		(*####################  DEBUG-MESSAGE  ###################################*)
		(*IF _debug_enable THEN
			LOG_CL.NEW_MSG := 'Repeat request after waittime / Part ~2 / Count ~3';
			LOG_CL.PRINTF[2] := INT_TO_STRING(cycle);
			LOG_CL.PRINTF[3] := USINT_TO_STRING(repeat_count);
			LOG_MSG();
		END_IF;*)
		(*########################################################################*)

		repeat_request := FALSE;
		state := 50;

	END_IF;

END_CASE;

(* ---------------- DNS --------------- *)
DNS_CLIENT(	IP_C:=IP_C,
			S_BUF:=S_BUF,
			R_BUF:=R_BUF,
			DOMAIN:=URL_DATA.DOMAIN,
			IP4_DNS:=DWORD#00,
			ACTIVATE:=state=40 (* DNS Start *)
			);
(* nicht oder nicht direkt verwendete Parameter *)
(*	DWORD :=DNS_CLIENT.IP4;
	BOOL  :=DNS_CLIENT.DONE;
	BYTE  :=DNS_CLIENT.ERROR; *)
(* -------------------------------------*)

(* ------------- HTTP_GET --------------- *)
HTTP_GET(	IP_C:=IP_C,
			S_BUF:=S_BUF,
			R_BUF:=R_BUF,
			IP4:=DNS_CLIENT.IP4,
			GET:=state=60,
			MODE:=BYTE#2, (* HTTP 1.1 mit persistenter Verbindung *)
			UNLOCK_BUF:=state=100,
			URL_DATA:=URL_DATA
			);

(* nicht oder nicht direkt verwendete Parameter *)
(*	STRING := HTTP_GET.HTTP_STATUS;
	UINT :=HTTP_GET.HEADER_START;
	UINT :=HTTP_GET.HEADER_STOP;
	UINT :=HTTP_GET.BODY_START;
	UINT :=HTTP_GET.BODY_STOP;
	BOOL :=HTTP_GET.DONE;
	BYTE :=HTTP_GET.ERROR;
*)
(* -------------------------------------*)

activate_last := ACTIVATE;

(*####################  DEBUG-MESSAGE  ###################################*)
(*IF _debug_enable THEN
	IF state <> _debug_state_last THEN
		LOG_CL.NEW_MSG := 'yw-step: /last ~1 /New ~2';
		LOG_CL.PRINTF[1] := INT_TO_STRING(_debug_state_last);
		LOG_CL.PRINTF[2] := INT_TO_STRING(state);
		LOG_MSG();
		_debug_state_last := state;
	END_IF;
END_IF;*)
(*########################################################################*)

(* revision history
ks	18. dez. 2008	rev 1.0
	original version

ks	01. oct. 2009	rev 1.1
	YAHOO_WEATHER_DATA

ks	24. sep. 2010	rev 1.2
	new URL-Location-parameter and REAL_CHECK (TwinCat BUG) 

ks	04. may. 2011	rev 1.3
	neue elemente:  CUR_CONDITIONS_ICON, FORCAST_TODAY_ICON, FORCAST_TOMORROW_ICON

ks	30. mar. 2016	rev 1.4
	änderung der api schnittstelle (URL) von yahoo

ks	01. jun. 2016	rev 1.5
	komplette überarbeitung auf neue yahoo-api

ks	22. may. 2017	rev 1.6
	automatische wiederholung der Abfrage wenn keine Daten vorhanden sind
*)

END_FUNCTION_BLOCK

// POUs/OTHER/XML_READER
FUNCTION_BLOCK XML_READER
VAR_IN_OUT
	CTRL : XML_CONTROL;
	BUF : NW_BUF_LONG;
END_VAR
VAR
	index :	INT;
	index2 : INT;
	stop : INT;
	mode : INT;
	command : WORD;
	c :	BYTE;
	s1 : INT;
	e1 : INT;
	path_overflow : BOOL;
	empty_tag : BOOL;
	s_code : STRING(10);
	e_code : STRING(10);
	watchdog : TON;

	(*LOG_MSG : LOG_MSG;
	_debug_enable : BOOL := TRUE;*)

END_VAR

(*

version 1.2		10. mai 2010
programmer 	ks
tested by		ks

XML_READER ermöglicht das serielle Parsen und die Auswertung von XML_Elementen in einem Buffer
*)

(*

TYP
00 = UNBEKANNT
01 = ELEMENT (STANDARD)
02 = CLOSE ELEMENT 
03 = TEXT
04 = ATTRIBUTE
05 = ELEMENT (PROCESSING INSTRUCTION) 

12 = !CDATA
13 = !COMMENT
14 = !DTD ELEMENT (Document Type Declarations )

98 = WATCHDOG
99 = ENDE

Bei Typ 02 werden keine Blockdaten ausgegeben !

*)

(* ---------- Init -------------- *)
IF OSCAT_BASIC.BIT_OF_DWORD(WORD_TO_DWORD(CTRL.COMMAND),15) THEN
	COMMAND := CTRL.COMMAND;
	CTRL.COMMAND := WORD#0;

	index := UINT_TO_INT(CTRL.START_POS);
	stop := UINT_TO_INT(CTRL.STOP_POS);
	mode := 100;
	path_overflow := FALSE;

	CTRL.TYP := 0;
	CTRL.COUNT := UINT#00;
	CTRL.LEVEL := UINT#00;
	CTRL.ATTRIBUTE := '';
	CTRL.ELEMENT := '';
	CTRL.PATH := '';
	CTRL.VALUE := '';

	WATCHDOG.PT := CTRL.WATCHDOG;
END_IF;

(*----------------------------------------------- *)

IF index < 0 THEN RETURN;END_IF;

CTRL.BLOCK1_START := UINT#0;
CTRL.BLOCK1_STOP := UINT#0;
CTRL.BLOCK2_START := UINT#0;
CTRL.BLOCK2_STOP := UINT#0;

WATCHDOG(IN:=FALSE); (* Timer stoppen *)

WHILE (TRUE) DO

	(* -------------- WATCHDOG ------------------ *)
	WATCHDOG(IN:=CTRL.WATCHDOG > T#0s);
	IF WATCHDOG.Q THEN
		CTRL.TYP := 98;
    		(*####################  DEBUG-MESSAGE  ###################################*)
    		(*IF _debug_enable THEN
      			LOG_CL.NEW_MSG := 'WATCHDOG:';
      			LOG_MSG();
    		END_IF;*)
    		(*########################################################################*)
		RETURN;
	END_IF;

	(* -------------- PARSING END ------------------ *)
	IF index > stop THEN
		CTRL.COUNT := CTRL.COUNT + UINT#1;
		CTRL.TYP := 99;
    		(*####################  DEBUG-MESSAGE  ###################################*)
    		(*IF _debug_enable THEN
      			LOG_CL.NEW_MSG := 'EX: #T:~1 #C:~2 #P:~6 #L:~7';
      			LOG_CL.PRINTF[1] := INT_TO_STRING(CTRL.TYP);
      			LOG_CL.PRINTF[2] := UINT_TO_STRING(CTRL.COUNT);
      			LOG_CL.PRINTF[6] := CTRL.PATH;
      			LOG_CL.PRINTF[7] := UINT_TO_STRING(CTRL.LEVEL);
      			LOG_MSG();
    		END_IF;*)
    		(*########################################################################*)
		mode  := 0; (* Schritt ruecksetzen *)
		index := 0; (* Abarbeitung stoppen *)
		RETURN;
	END_IF;

	CASE mode OF

	100: (* ---------- ELEMENT SECTION ------------------ *)
		(* search begin of element *)
		s1 := 0;
		e1 := 0;
		WHILE (index <= stop) DO
			IF BUF[INDEX]=BYTE#60 THEN (* '<' TagBegin *)
				index := index + 1;
				C := BUF[index];
				IF C = BYTE#47 THEN (* '/' TagTerm *)
					mode := 300; (* End Element Section *)
				ELSIF C = BYTE#33 THEN (* '!' for Special Section *)
					index := index + 1;
					mode := 500;
				ELSE
					s1 := index;
				END_IF;
				EXIT;
			END_IF;
			index := index + 1;
		END_WHILE;

		(* analyse element *)
		CTRL.TYP := 0; (* TYP löschen *)
		IF s1 > 0 THEN
			WHILE (index <= stop AND e1 = 0) DO
				c := BUF[index];
				(* whitespace zeichen = Element with Attributes *)
				IF c <= BYTE#32 THEN
					(* suche nächstes druckbares zeichen *)
					index2 := index;
					WHILE (index2 <= stop) AND (BUF[index2] <= BYTE#32) DO
						index2 := index2 + 1;
					END_WHILE;
					IF BUF[index2] = BYTE#47 THEN (* pruefe auf leeres Element '/' *)
						index := index2;
						e1 := index - 2;
						CTRL.TYP := 1; (* struktur-element *)
						mode := 300;   (* Close Element *)
						EXIT;
					END_IF;

					e1 := index - 1;
					CTRL.TYP := 1; (* Element mit Attribute *)
					mode := 400;

				ELSIF c = BYTE#62 THEN (* '>' TagEnd *)

					(* pruefe auf leeres Element <xx/> *)
					index2 := index - 1;
					IF BUF[index2] = BYTE#47 THEN (* TagTerm '/' *)
						e1 := index2 - 1;
						CTRL.TYP := 1;
						EMPTY_TAG := TRUE; (* EMPTY TAG Mode *)
						mode := 200; (* TEXT Element *)
						EXIT;
					END_IF;

					e1 := index - 1;
					index2 := index + 1;

					(* untersuche nachfolgendes Element *)
					WHILE (index2 <= stop) DO
						c := BUF[index2];
						IF c = BYTE#60 THEN (* '<' TagBegin *)

							index2 := index2 + 1; (* geht bei PCWORX leider nicht anders !*)
							c := BUF[index2];
							index2 := index2 - 1;
							IF c = BYTE#47 THEN (* TagTerm '/' *)
								empty_tag := TRUE;
								mode := 200; (* TEXT Element *)
							ELSE
								mode := 100; (* Element *)
							END_IF;
							CTRL.TYP := 1; (* struktur-element *)
							EXIT;
						ELSIF c > BYTE#32  THEN (* Printable-Character *)
							CTRL.TYP := 1; (* element with text *)
							mode := 200;
							EXIT;
						END_IF;
						index2 := index2 + 1;
					END_WHILE;
				END_IF;
				index := index + 1;
			END_WHILE;
		END_IF;

		(* Neues Element gefunden*)
		IF CTRL.TYP > 0 THEN

			(* Sonderprüfung auf Processing Instruction (PI) *)
			IF BUF[s1] = BYTE#63 THEN (* '?' for Processing Instruction *)
				s1 := s1 + 1; (* führendes '?' auslassen *)
				CTRL.TYP := 5;
			END_IF;
			CTRL.BLOCK1_START := INT_TO_UINT(s1);
			CTRL.BLOCK1_STOP  := INT_TO_UINT(e1);
			CTRL.ELEMENT := OSCAT_BASIC.BUFFER_TO_STRING(PT:=ADR(BUF),SIZE:=INT_TO_UINT(stop + 1),START:=CTRL.BLOCK1_START,STOP:=CTRL.BLOCK1_STOP);
			CTRL.COUNT := CTRL.COUNT + UINT#1;
			CTRL.LEVEL := CTRL.LEVEL + UINT#1;

			IF path_overflow = FALSE THEN
				(* Stringlänge überwachen *)
				IF LEN(CTRL.PATH) + LEN(CTRL.ELEMENT) + 1 > 250 THEN
					path_overflow := TRUE;
					CTRL.PATH := 'OVERFLOW';
				ELSE
					CTRL.PATH := CONCAT(CTRL.PATH,'/');
					CTRL.PATH  := CONCAT(CTRL.PATH,CTRL.ELEMENT);
				END_IF;
			END_IF;

			IF OSCAT_BASIC.BIT_OF_DWORD(WORD_TO_DWORD(COMMAND),CTRL.TYP) THEN
        				(*####################  DEBUG-MESSAGE  ###################################*)
        				(*IF _debug_enable THEN
          				LOG_CL.NEW_MSG := 'EL: #T:~1 #C:~2 #E:~3 #P:~6 #L:~7';
          				LOG_CL.PRINTF[1] := INT_TO_STRING(CTRL.TYP);
          				LOG_CL.PRINTF[2] := UINT_TO_STRING(CTRL.COUNT);
          				LOG_CL.PRINTF[3] := CTRL.ELEMENT;
          				LOG_CL.PRINTF[6] := CTRL.PATH;
          				LOG_CL.PRINTF[7] := UINT_TO_STRING(CTRL.LEVEL);
          				LOG_MSG();
        				END_IF;*)
        				(*########################################################################*)
				RETURN;
			END_IF;
		END_IF;

	200: (* ---------- TEXT SECTION ------------------ *)
		CTRL.VALUE := '';
		IF empty_tag = FALSE THEN
			s1 := index;
			(* suche '<' EndTag*)
			WHILE (index <= stop) AND (BUF[index] <> BYTE#60) DO
				index := index + 1;
			END_WHILE;

			E1 := index - 1;
			CTRL.BLOCK1_START := INT_TO_UINT(s1);
			CTRL.BLOCK1_STOP  := INT_TO_UINT(e1);
			CTRL.VALUE := OSCAT_BASIC.BUFFER_TO_STRING(PT:=ADR(BUF),SIZE:=INT_TO_UINT(stop + 1),START:=CTRL.BLOCK1_START,STOP:=CTRL.BLOCK1_STOP);
		END_IF;

		empty_tag := FALSE;
		mode := 300; (* -> NEXT-JOB: END ELEMENT *)
		CTRL.COUNT := CTRL.COUNT + UINT#1;
		CTRL.TYP := 3;

		IF OSCAT_BASIC.BIT_OF_DWORD(WORD_TO_DWORD(command),CTRL.TYP) THEN
      			(*####################  DEBUG-MESSAGE  ###################################*)
      			(*IF _debug_enable THEN
        				LOG_CL.NEW_MSG := 'TE: #T:~1 #C:~2 #E:~3 #V:~4 #P:~6 #L:~7';
        				LOG_CL.PRINTF[1] := INT_TO_STRING(CTRL.TYP);
        				LOG_CL.PRINTF[2] := UINT_TO_STRING(CTRL.COUNT);
        				LOG_CL.PRINTF[3] := CTRL.ELEMENT;
        				LOG_CL.PRINTF[4] := CTRL.VALUE;
        				LOG_CL.PRINTF[6] := CTRL.PATH;
        				LOG_CL.PRINTF[7] := UINT_TO_STRING(CTRL.LEVEL);
        				LOG_MSG();
      			END_IF;*)
      			(*########################################################################*)
			RETURN;
		END_IF;

	300: (* ---------- END ELEMENT SECTION ------------------ *)
		WHILE (index <= stop) DO
			c := BUF[index];
			IF c = BYTE#62 THEN (* '>' TagEnd *)
				index := index + 1;
				s1 := OSCAT_BASIC.FINDB(str1:=CTRL.PATH,str2:='/');
				IF path_overflow = FALSE THEN
					IF s1 > 1 THEN
						CTRL.ELEMENT := RIGHT(CTRL.PATH,LEN(CTRL.PATH) - s1);
						CTRL.PATH := LEFT(CTRL.PATH,s1 - 1);
					ELSE
						CTRL.ELEMENT := RIGHT(CTRL.PATH,LEN(CTRL.PATH) - 1);
						CTRL.PATH :='';
					END_IF;
				END_IF;

				CTRL.LEVEL := CTRL.LEVEL - UINT#1;
				CTRL.COUNT := CTRL.COUNT + UINT#1;
				CTRL.TYP := 2;
				mode := 100;

				IF OSCAT_BASIC.BIT_OF_DWORD(WORD_TO_DWORD(COMMAND),CTRL.TYP) THEN
         	 				(*####################  DEBUG-MESSAGE  ###################################*)
          				(*IF _debug_enable THEN
            					LOG_CL.NEW_MSG := 'CE: #T:~1 #C:~2 #E:~3 #P:~6 #L:~7';
            					LOG_CL.PRINTF[1] := INT_TO_STRING(CTRL.TYP);
            					LOG_CL.PRINTF[2] := UINT_TO_STRING(CTRL.COUNT);
            					LOG_CL.PRINTF[3] := CTRL.ELEMENT;
            					LOG_CL.PRINTF[6] := CTRL.PATH;
            					LOG_CL.PRINTF[7] := UINT_TO_STRING(CTRL.LEVEL);
            					LOG_MSG();
          				END_IF;*)
          				(*########################################################################*)
					RETURN;
				ELSE
					EXIT;
				END_IF;
			END_IF;
			index := index + 1;
		END_WHILE;

	400: (* ---------- ATTRIBUTE SECTION ------------------ *)
		(* search first normal charakter *)
		WHILE (index <= stop AND BUF[index] <= BYTE#32) DO
			index := index + 1;
		END_WHILE;

		(* begin Attribe name *)
		e1 := 0;
		s1 := index;
		(* search end of Attrib Name '=' *)
		WHILE (index <= stop) DO
			IF BUF[index] = BYTE#61 THEN (* '=' Equals *)
				e1 := index - 1;
				EXIT;
			END_IF;
			index := index + 1;
		END_WHILE;

		IF e1 > 0 THEN
			(* Attribute Name *)
			CTRL.BLOCK1_START := INT_TO_UINT(s1);
			CTRL.BLOCK1_STOP  := INT_TO_UINT(e1);
			CTRL.ATTRIBUTE := OSCAT_BASIC.BUFFER_TO_STRING(PT:=ADR(BUF),SIZE:=INT_TO_UINT(STOP + 1),START:=CTRL.BLOCK1_START,STOP:=CTRL.BLOCK1_STOP);
			(* search end of Attrib Value '=' *)
			index := index + 2;
			e1 := 0;
			s1 := INDEX;
			WHILE (index <= stop AND e1 = 0) DO
				c := BUF[index];
				IF c = BYTE#34 OR c = BYTE#39 THEN (* " OR ' Equals *)
					e1 := index - 1;
				END_IF;
				index := index + 1;
			END_WHILE;

			IF e1 > 0 THEN
				(* Value *)
				CTRL.BLOCK2_START := INT_TO_UINT(s1);
				CTRL.BLOCK2_STOP  := INT_TO_UINT(e1);

				(* bei leeren "" ist start groesser als stop und wird somit zum leerstring *)
				CTRL.VALUE := OSCAT_BASIC.BUFFER_TO_STRING(PT:=ADR(BUF),SIZE:=INT_TO_UINT(stop + 1),START:=CTRL.BLOCK2_START,STOP:=CTRL.BLOCK2_STOP);
				(* search next non white space charakter *)
				WHILE (index <= stop AND BUF[index] <= BYTE#32) DO
					index := index + 1;
				END_WHILE;

					c := BUF[index];
					(* TagEnd '>' *)
					IF c = BYTE#62 THEN
						index := index + 1;
						index2 := index;

					(* search next non white space charakter *)
					WHILE (index <= stop AND BUF[index] <= BYTE#32) DO
						index := index + 1;
					END_WHILE;

					IF BUF[index] = BYTE#60 THEN (* TagBegin '<' *)
						mode := 100; (* -> NEXT-JOB: ELEMENT-SECTION *)
					ELSE
						index := index2;
						mode := 200; (* -> NEXT-JOB: TEXT-SECTION *)
					END_IF;

				ELSIF c = BYTE#47 OR c = BYTE#63 THEN (* TagTerm '/' OR '?' end Processing Instruction *)
					mode := 300; (* -> NEXT-JOB: END ELEMENT *)
				ELSE
					mode := 400; (* -> NEXT-JOB: ATTRIBUTE-SECTION *)
				END_IF;

				CTRL.COUNT := CTRL.COUNT + UINT#1;
				CTRL.TYP := 4;
				IF OSCAT_BASIC.BIT_OF_DWORD(WORD_TO_DWORD(command),CTRL.TYP) THEN
          				(*####################  DEBUG-MESSAGE  ###################################*)
          				(*IF _debug_enable THEN
            					LOG_CL.NEW_MSG := 'AT: #T:~1 #C:~2 #E:~3 #A:~4 #V:~5 #P:~6 #L:~7';
            					LOG_CL.PRINTF[1] := INT_TO_STRING(CTRL.TYP);
            					LOG_CL.PRINTF[2] := UINT_TO_STRING(CTRL.COUNT);
            					LOG_CL.PRINTF[3] := CTRL.ELEMENT;
            					LOG_CL.PRINTF[4] := CTRL.ATTRIBUTE;
            					LOG_CL.PRINTF[5] := CTRL.VALUE;
            					LOG_CL.PRINTF[6] := CTRL.PATH;
            					LOG_CL.PRINTF[7] := UINT_TO_STRING(CTRL.LEVEL);
            					LOG_MSG();
          				END_IF;*)
          				(*########################################################################*)
					RETURN;
				END_IF;
			END_IF;
		END_IF;

	500: (* ---------- SPECIAL DATA SECTION (Document Type Declarations) ---------- *)

		CTRL.TYP := 0;
		s1 := 0;
		index2 := 11;

		WHILE (s1 = 0) DO
			index2 := index2 + 1;
			CTRL.TYP := index2;

			CASE index2 OF
			12: (* CDATA *)
				s_code := '[CDATA[';
				e_code := ']]>';
			13: (* COMMENT *)
				s_code := '--';
				e_code := '-->';
			14: (* ANY DTD *)
				e_code := '';
				s1 := index;
				EXIT;
			END_CASE;

			e1 := LEN(s_code);
			IF OSCAT_BASIC.BUFFER_SEARCH(PT:=ADR(BUF),SIZE:=INT_TO_UINT(index + e1),STR:=S_CODE,POS:=index,IGN:=FALSE) = INDEX THEN
				s1 := index + e1;
			END_IF;
		END_WHILE;

		CTRL.BLOCK1_START := INT_TO_UINT(s1);
		IF LEN(e_code) > 0 THEN
			(* Ende Kennung suchen *)
			e1 := OSCAT_BASIC.BUFFER_SEARCH(PT:=ADR(BUF),SIZE:=INT_TO_UINT(stop + 1),STR:=e_code,POS:=index,IGN:=FALSE);
			CTRL.BLOCK1_STOP := INT_TO_UINT(e1 - 1);
			index := e1 + LEN(e_code); (* naechstes element *)
		ELSE
			(* suche '>' EndTag*)
			index2 := 1; (* <> Paar zähler *)
			WHILE (index <= stop AND index2 > 0) DO
				c := BUF[index];
				IF c = BYTE#60 THEN (* '<' TagBegin *)
					index2 := index2 + 1;
				ELSIF c = BYTE#62 THEN (* '>' TagEnd   *)
					index2 := index2 - 1;
				ELSIF c = BYTE#34 OR c = BYTE#39 THEN (* " Double Quote OR ' Single Quote *)
					index := index + 1;
					WHILE (index <= stop) DO
						c := BUF[index];
						IF c = BYTE#34 OR c = BYTE#39 THEN (* " Double Quote OR ' Single Quote *)
							EXIT;
						END_IF;
						index := index + 1;
					END_WHILE;
				END_IF;
				index := index + 1;
			END_WHILE;
			CTRL.BLOCK1_STOP := INT_TO_UINT(index - 2);
		END_IF;

		CTRL.VALUE := OSCAT_BASIC.BUFFER_TO_STRING(PT:=ADR(BUF),SIZE:=INT_TO_UINT(stop + 1),START:=CTRL.BLOCK1_START,STOP:=CTRL.BLOCK1_STOP);
		CTRL.COUNT := CTRL.COUNT + UINT#1;
		mode := 100; (* -> NEXT-JOB: ELEMENT *)

		IF OSCAT_BASIC.BIT_OF_DWORD(WORD_TO_DWORD(command),CTRL.TYP) THEN
      			(*####################  DEBUG-MESSAGE  ###################################*)
      			(*IF _debug_enable THEN
        				LOG_CL.NEW_MSG := 'DTD: #T:~1 #C:~2 #S:~3 #E:~4 #V:~5 #P:~6 #L:~7';
        				LOG_CL.PRINTF[1] := INT_TO_STRING(CTRL.TYP);
        				LOG_CL.PRINTF[2] := UINT_TO_STRING(CTRL.COUNT);
        				LOG_CL.PRINTF[3] := UINT_TO_STRING(CTRL.BLOCK1_START);
        				LOG_CL.PRINTF[4] := UINT_TO_STRING(CTRL.BLOCK1_STOP);
        				LOG_CL.PRINTF[5] := CTRL.VALUE;
        				LOG_CL.PRINTF[6] := CTRL.PATH;
        				LOG_CL.PRINTF[7] := UINT_TO_STRING(CTRL.LEVEL);
        				LOG_MSG();
      			END_IF;*)
      			(*########################################################################*)
			RETURN;
		END_IF;

	END_CASE;
END_WHILE;


(* revision history
ks	18. oct. 2008	rev 1.0
	original version

ks	20. oct. 2009	rev 1.1
	Networkbuffer und Buffer-funktionen auf Basis 0

ks	10. mai. 2010	rev 1.2
	stringlänge maximal 250 zeichen

*)

END_FUNCTION_BLOCK

// POUs/DEMO/DNS_DYN_DEMO
PROGRAM DNS_DYN_DEMO
VAR
	DNS_DYN : DNS_DYN;
	IP_C : IP_C;
	S_BUF : NETWORK_BUFFER;
	R_BUF : NETWORK_BUFFER;
	IP_CONTROL : IP_CONTROL;
	enable: BOOL;
	done : BOOL;
	error_c : DWORD;
	error_t : BYTE;
	busy : BOOL;
	COUNT_DR: oscat_basic.COUNT_DR;
	z: DWORD;

	GET_WAN_IP : GET_WAN_IP;
	t1: TON;
	done2 : BOOL;
	error_c2 : DWORD;
	error_t2 : BYTE;
	update : BOOL;
	new_ip: BOOL;
	wan_ip4: DWORD;
END_VAR
VAR // added by the converter: edge detectors and wires of the graphical bodies
    _w1 : ANY;
END_VAR

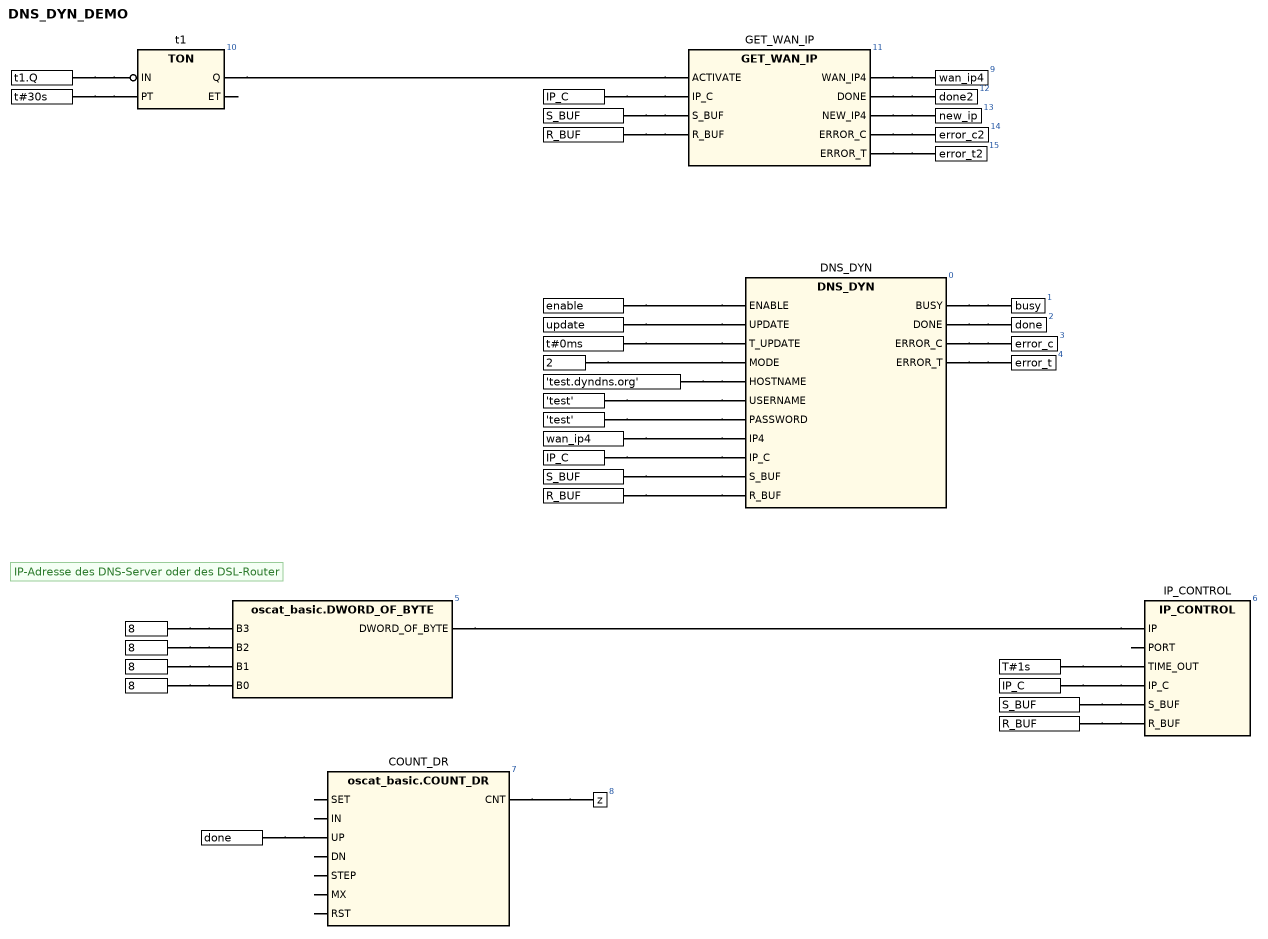
DNS_DYN(
    ENABLE := enable,
    UPDATE := update,
    T_UPDATE := t#0ms,
    MODE := 2,
    HOSTNAME := 'test.dyndns.org',
    USERNAME := 'test',
    PASSWORD := 'test',
    IP4 := wan_ip4,
    IP_C := IP_C,
    S_BUF := S_BUF,
    R_BUF := R_BUF);
busy := DNS_DYN.BUSY;
done := DNS_DYN.DONE;
error_c := DNS_DYN.ERROR_C;
error_t := DNS_DYN.ERROR_T;
// IP-Adresse des DNS-Server oder des DSL-Router
_w1 := oscat_basic.DWORD_OF_BYTE(B3 := 8, B2 := 8, B1 := 8, B0 := 8);
IP_CONTROL(IP := _w1, TIME_OUT := T#1s, IP_C := IP_C, S_BUF := S_BUF, R_BUF := R_BUF);
COUNT_DR(UP := done); // oscat_basic.COUNT_DR
z := COUNT_DR.CNT;
wan_ip4 := GET_WAN_IP.WAN_IP4;
t1(IN := NOT t1.Q, PT := t#30s); // TON
GET_WAN_IP(ACTIVATE := t1.Q, IP_C := IP_C, S_BUF := S_BUF, R_BUF := R_BUF);
done2 := GET_WAN_IP.DONE;
new_ip := GET_WAN_IP.NEW_IP4;
error_c2 := GET_WAN_IP.ERROR_C;
error_t2 := GET_WAN_IP.ERROR_T;

END_PROGRAM

// POUs/NETWORK/GET_WAN_IP
FUNCTION_BLOCK GET_WAN_IP
VAR_IN_OUT
	IP_C : IP_C; (* IP_Control Verwaltungsstruktur *)
	S_BUF : NETWORK_BUFFER;
	R_BUF : NETWORK_BUFFER;
END_VAR
VAR_INPUT
	ACTIVATE : BOOL;
END_VAR
VAR_OUTPUT
	WAN_IP4 : DWORD;
	DONE : BOOL;
	NEW_IP4 : BOOL;
	ERROR_C : DWORD;
	ERROR_T : BYTE;
END_VAR
VAR
	URL_DATA : url;
	DNS_CLIENT : DNS_CLIENT;
	HTTP_GET : HTTP_GET;
	activate_last : BOOL;
	wan_ip4_last : DWORD;
	state : INT;
	st_ip : STRING(120);
	i1 :	INT;
	p1 : INT;
	p2 : INT;
	p3 : INT;
END_VAR

(*
version 1.1	28. dec. 2009
programmer 	ks
tested by	ks

GET_WAN_IP ermittelt die aktuelle WAN-IP (Internet-Adresse)
*)

CASE state OF

00:
	IF ACTIVATE AND NOT activate_last THEN
		state := 20;
		DONE := FALSE;
		ERROR_C := DWORD#0;
		ERROR_T := BYTE#0;
	END_IF;

20: (* URL for DNS UND HTTP-GET *)
	URL_DATA := STRING_TO_URL(STR:='checkip.dyndns.com',DEFAULT_PROTOCOL:='',DEFAULT_PATH:='');
	state := 40;

40:
	IF DNS_CLIENT.DONE THEN
		state := 60;
	ELSIF (DNS_CLIENT.ERROR > DWORD#00) THEN
		(* Fehlerbehandlung *)
		ERROR_C := DNS_CLIENT.ERROR;
		ERROR_T := BYTE#01;
		state := 100;
	END_IF;

60:
	IF HTTP_GET.DONE THEN
		state := 80;
	ELSIF (HTTP_GET.ERROR > DWORD#00) THEN
		(* Fehlerbehandlung *)
		ERROR_C := HTTP_GET.ERROR;
		ERROR_T := BYTE#02;
		state := 100;
	END_IF;

80:
	(* Als Antwort wird folgende HTML Seite empfangen , hier muss die IP-Adresse herauskopiert werden *)
	(* <html><head><title>Current IP Check</title></head><body>Current IP Address: 85.127.217.33</body></html> *)
	st_ip := '';
	p1 := 0;
	FOR i1 := UINT_TO_INT(HTTP_GET.BODY_START) TO UINT_TO_INT(HTTP_GET.BODY_STOP) DO
		IF R_BUF.BUFFER[i1] = BYTE#58 THEN (* suche ':' *)
			p1 := i1 + 2;
			EXIT;
		END_IF;
	END_FOR;

	p3 := p1 + 15;
	IF p1 > 0 AND p3 < UINT_TO_INT(HTTP_GET.BODY_STOP) THEN
		FOR p2 := p1 TO p3 DO
			IF R_BUF.BUFFER[p2] <> BYTE#60 THEN (* suche '<' *)
				st_ip := CONCAT(st_ip,OSCAT_BASIC.CHR_TO_STRING(C:=R_BUF.BUFFER[p2]));
			ELSE
				EXIT;
			END_IF;
		END_FOR;
	END_IF;

	WAN_IP4 := IP4_DECODE(STR:=st_ip);

	IF WAN_IP4 <> DWORD#0 THEN
		DONE := TRUE;
		NEW_IP4 := WAN_IP4 <> wan_ip4_last;
		wan_ip4_last := WAN_IP4;
	ELSE
		ERROR_C := DWORD#01; (* keine gültige IP gefunden *)
		ERROR_T := BYTE#03;
	END_IF;
	state := 100;

100:
	(* UNLOCK HTTP DATA *)
	IF (NOT HTTP_GET.DONE) THEN
		state := 0;
		DONE := ERROR_T = BYTE#0;
	END_IF;

END_CASE;

(* ---------------- DNS --------------- *)
DNS_CLIENT(	IP_C:=IP_C,
			S_BUF:=S_BUF,
			R_BUF:=R_BUF,
			DOMAIN:=URL_DATA.DOMAIN,
			IP4_DNS:=DWORD#00,
			ACTIVATE:=state=40 (* DNS Start *)
			);
(* nicht oder nicht direkt verwendete Parameter *)
(* DWORD :=DNS_CLIENT.IP4;
   BOOL  :=DNS_CLIENT.DONE;
   BYTE  :=DNS_CLIENT.ERROR; *)
(* -------------------------------------*)

(* ------------- HTTP_GET --------------- *)

HTTP_GET(	IP_C:=IP_C,
			S_BUF:=S_BUF,
			R_BUF:=R_BUF,
			IP4:=DNS_CLIENT.IP4,
			GET:=state=60,
			MODE:=BYTE#2, (* HTTP 1.1 mit persistenter Verbindung *)
			UNLOCK_BUF:=state=100,
			URL_DATA:=URL_DATA
			);

(* nicht oder nicht direkt verwendete Parameter *)
(*STRING := HTTP_GET.HTTP_STATUS;
  UINT :=HTTP_GET.HEADER_START;
  UINT :=HTTP_GET.HEADER_STOP;
  UINT :=HTTP_GET.BODY_START;
  UINT :=HTTP_GET.BODY_STOP;
  BOOL :=HTTP_GET.DONE;
  BYTE :=HTTP_GET.ERROR;
*)
(* -------------------------------------*)

activate_last := ACTIVATE;

(* revision history
ks	28. dec 2009	rev 1.1
	original version

*)

END_FUNCTION_BLOCK

// POUs/NETWORK/DNS_REV_CLIENT
FUNCTION_BLOCK DNS_REV_CLIENT
VAR_IN_OUT
	IP_C : IP_C; (* IP_Control Verwaltungsstruktur *)
	S_BUF : NETWORK_BUFFER;
	R_BUF : NETWORK_BUFFER;
END_VAR
VAR_INPUT
	ACTIVATE : BOOL;
	IP4 : DWORD;
	IP4_DNS : DWORD;
END_VAR
VAR_OUTPUT
	DOMAIN : STRING;
	DONE : BOOL;
	ERROR : DWORD;
END_VAR
VAR
	IP_FIFO : IP_FIFO;
	ip_state : BYTE;
	ip_id : BYTE;
	state : INT;
	ip4_copy : DWORD;
	d : STRING(27);
	activate_last : BOOL;
	i : INT;
	dl : INT;
	p1 : INT;
	char : BYTE;
	char_count : INT;
	tid : BYTE;
END_VAR

(*
version 1.0	28. dec. 2009
programmer 	ks
tested BY	ks

DNS_REV_CLIENT führt eine Reverse-Domain-Name Abfrage durch, und ermittelt aus einer IP-Adresse den zugehörigen Domain-Namen.

*)

(* Domain Name System (query) *)

CASE state OF
00: (* auf positive Flanke GET warten *)
	IF ACTIVATE AND NOT activate_last THEN
		ERROR := DWORD#0;
		ip4_copy := ip4; (* IP4 sichern *)
		ip_state := BYTE#1;
		DOMAIN := '';
		DONE := FALSE;

		d := '';
		FOR i := 1 TO 4 DO
			d := CONCAT(d,BYTE_TO_STRING(DWORD_TO_BYTE(IP4)));
			d := CONCAT(d,'.');
			IP4 := ROR(IP4,8);
		END_FOR;
		d := CONCAT(d,'in-addr.arpa');
		state := 10;
	END_IF;

10: (* Bei IP_Control anmelden *)
	IF ip_state = BYTE#3 THEN
		dl := LEN(d);

		(* sendebuffer initialisieren *)
		char_count := 17 + dl;
		FOR i := 0 TO char_count DO
			S_BUF.BUFFER[i] := BYTE#00;
		END_FOR;

		tid := UINT_TO_BYTE(BYTE_TO_UINT(tid) + UINT#1);
		S_BUF.BUFFER[01] := tid; (* Transaction ID lowbyte *)
		S_BUF.BUFFER[02] := BYTE#16#01; (* Flags: highbyte *)
		S_BUF.BUFFER[05] := BYTE#16#01; (* Questions: lowbyte *)

		(* den servernamen von hinten nach vorne bearbeiten *)
		i := dl + 12;
		char_count := 0;

		WHILE i > 12 DO
			char := OSCAT_BASIC.CODE(STR:=d,POS:=i - 12);

			(* prüfe auf haupt/sub domänen namens-teiler "." *)
			IF char = BYTE#46 THEN
				(* anstelle des teilers "." wird die länge des erkannten haupt/sub domänennames eingetragen *)
				S_BUF.BUFFER[i] := INT_TO_BYTE(char_count);
				char_count := 0;
			ELSE
				S_BUF.BUFFER[i] := char; (* char in buffer eintragen *)
				char_count := char_count + 1; (* anzahl char zählen *)
			END_IF;
			i := i - 1;
		END_WHILE;

		S_BUF.BUFFER[i] := INT_TO_BYTE(char_count); (* längenangabe des ganz linken (ersten) domänennamens eintragen *)
		i := dl + 15; (* position hinter dem servernamen *)
		S_BUF.BUFFER[i] := BYTE#12; (* Type: PTR (Domain name pointer) lowbyte *)
		i := i + 2;
		S_BUF.BUFFER[i] := BYTE#01; (* Class: IN lowbyte *)
		i := i + 1;

		(* IP Datenverkehr einrichten *)
		IP_C.C_PORT := WORD#53; (* Portnummer eintragen *)
		IP_C.C_IP := IP4_DNS; (* IP eintragen *)
		IP_C.C_MODE := BYTE#1; (* Mode: UDP+AKTIV+PORT+IP *)
		IP_C.C_ENABLE := TRUE; (* Verbindungsaufbau freigeben *)
		IP_C.TIME_RESET := TRUE; (* Zeitueberwachung rücksetzen *)
		IP_C.R_OBSERVE  := TRUE; (* Datenempfang ueberwachen *)
		S_BUF.SIZE := INT_TO_UINT(i); (* sendelänge eintragen *)
		R_BUF.SIZE := UINT#0; (* Empfangslänge rücksetzen *)
		state := 30;
	END_IF;

30:
	IF IP_C.ERROR <> DWORD#00 THEN
		ERROR := IP_C.ERROR;
	(* prüfe ob antwort telegramm die richtige Transaction-ID und mindestlänge hat *)
	ELSIF (S_BUF.SIZE = UINT#0) AND (tid = R_BUF.BUFFER[1]) AND (R_BUF.SIZE >= INT_TO_UINT(i+12)) THEN

		(* prüfe Return code der Flags. 4 bits *)
		ERROR := BYTE_TO_DWORD(R_BUF.BUFFER[3] AND BYTE#2#0000_1111);

		IF ERROR = DWORD#00 THEN

			i := R_BUF.SIZE - 2;
			WHILE R_BUF.BUFFER[i] > 0 DO
				IF i = 0 THEN EXIT; END_IF;
				i := i - 1;
			END_WHILE;

			i := i + 2;
			p1 := i + 1;
			WHILE i < R_BUF.SIZE DO
				dl := R_BUF.BUFFER[i];
				IF dl > 0 THEN
					R_BUF.BUFFER[i] := BYTE#46;
					i := i + dl + 1;
				ELSE
					DOMAIN := OSCAT_BASIC.BUFFER_TO_STRING(PT:=ADR(R_BUF.BUFFER),SIZE:=SIZEOF(R_BUF.BUFFER),START:=p1,STOP:=i-1);
					EXIT;
				END_IF;
			END_WHILE;
			state := 0;
			DONE := TRUE;
		END_IF;
	END_IF;

	IF ERROR <> DWORD#0 THEN
		state := 0;
	END_IF;

	IF state = 0 THEN
		IP_C.R_OBSERVE := FALSE; (* Datenempfang ueberwachen *)
		ip_state := BYTE#4; (* Abmelden *)
	END_IF;

END_CASE;

activate_last := ACTIVATE; (* letzten Status sichern zur Flankenerkennung *)

(* IP_FIFO *)
IP_FIFO(FIFO:=IP_C.FIFO,STATE:=ip_state,ID:=ip_id);

(* revision history

ks	28. dec. 2009	rev 1.0
	original version

*)


(*----------------------------------------------------------------------------------------------------------------*)
(* Flags: 0x0100 (Standard query)                                                                                            *)
(* 0... .... .... .... = Response: Message is a query                                                                   *)
(* .000 0... ....  = Opcode: Standard query (0)                                                                          *)
(* .... ..0. .... .... = Truncated: Message is not truncated                                                          *)
(* .... ...1 .... .... = Recursion desired: Do query recursively                                                    *)
(* .... .... .0.. .... = Z: reserved (0)                                                                                                  *)
(* .... .... ...0 .... = Non-authenticated data OK: Non-authenticated data is unacceptable *)
(*-----------------------------------------------------------------------------------------------------------------*)

(*
Errorcodes  Description	References 
000	No error. 		 	The request completed successfully.
001	Format error. 		The name server was unable to interpret the query. 
002	Server failure.  	The name server was unable to process this query due to a problem with the name server. 
003	Name Error. 	 	Meaningful only for responses from an authoritative name server, this code signifies that the domain name referenced in the query does not exist.
004	Not Implemented. 	The name server does not support the requested kind of query.
005	Refused. 			The name server refuses to perform the specified operation for policy reasons.
  						 For example, a name server may not wish to provide the information to the particular requester, or a name server may not wish to perform a particular operation (e.g., zone transfer) for particular data.
006	YXDomain.			Name Exists when it should not. 
007	YXRRSet. RR			Set Exists when it should not. 
008	NXRRSet. RR			Set that should exist does not. 
009	NotAuth.			Server Not Authoritative for zone. 
010	NotZone,			Name not contained in zone. 
255	Timeout				No Response  
*)

END_FUNCTION_BLOCK

// POUs/DEMO/DNS_REV_DEMO
PROGRAM DNS_REV_DEMO
VAR
	DNS_REV_CLIENT: DNS_REV_CLIENT;
	IP_C : IP_C;
	S_BUF : NETWORK_BUFFER;
	R_BUF : NETWORK_BUFFER;
	IP_CONTROL : IP_CONTROL;
	activate : BOOL := TRUE;
	done : BOOL;
	error: DWORD;
	domain: STRING;
END_VAR
VAR // added by the converter: edge detectors and wires of the graphical bodies
    _w1, _w2 : ANY;
END_VAR

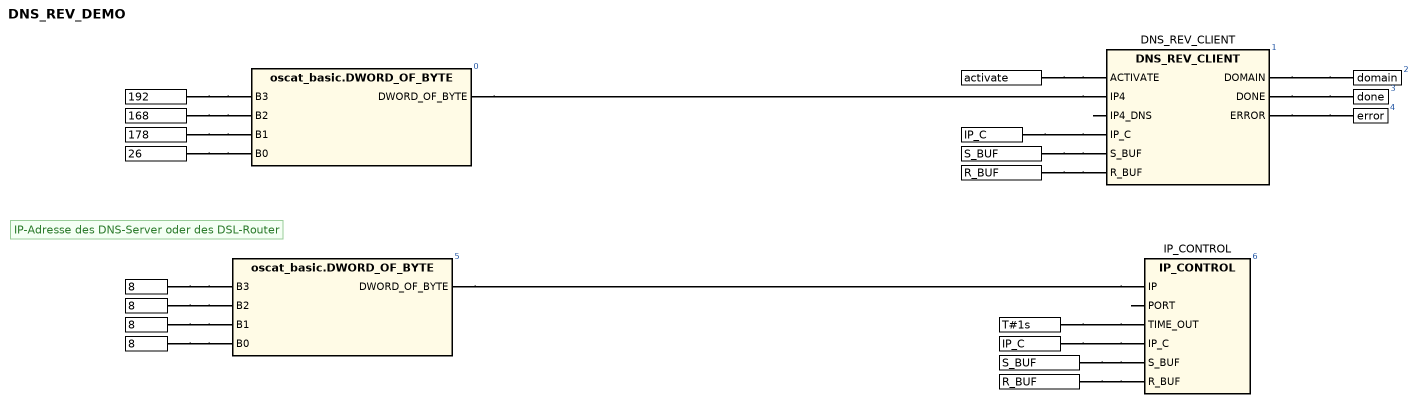
_w1 := oscat_basic.DWORD_OF_BYTE(B3 := 192, B2 := 168, B1 := 178, B0 := 26);
DNS_REV_CLIENT(ACTIVATE := activate, IP4 := _w1, IP_C := IP_C, S_BUF := S_BUF, R_BUF := R_BUF);
domain := DNS_REV_CLIENT.DOMAIN;
done := DNS_REV_CLIENT.DONE;
error := DNS_REV_CLIENT.ERROR;
// IP-Adresse des DNS-Server oder des DSL-Router
_w2 := oscat_basic.DWORD_OF_BYTE(B3 := 8, B2 := 8, B1 := 8, B0 := 8);
IP_CONTROL(IP := _w2, TIME_OUT := T#1s, IP_C := IP_C, S_BUF := S_BUF, R_BUF := R_BUF);

END_PROGRAM

// POUs/DEMO/DNS_SNTP_SYSLOG_DEMO
PROGRAM DNS_SNTP_SYSLOG_DEMO
VAR
	IP_C : IP_C;
	S_BUF : NETWORK_BUFFER;
	R_BUF : NETWORK_BUFFER;
	IP_CONTROL_1: IP_CONTROL;
	DNS_CLIENT : DNS_CLIENT;
	SNTP_CLIENT: SNTP_CLIENT;
	SNTP_SERVER: SNTP_SERVER;
	COUNT_DR: oscat_basic.COUNT_DR;
	RTC_2: oscat_basic.RTC_2;
	count_cycles: DWORD;
	dns_error: DWORD;
	sntp_error: DWORD;
	freigabe: BOOL;
	dso: BOOL;
	xms: INT;
	sntp_srv_enable: BOOL;
	cur_UDT: DT;
	cur_LOC_DT: DT;
	SYS_LOG: SYS_LOG;
	sys_log_option: BYTE := 2#0000_0100;
	TON_1: TON;
	tp_sys_log: BOOL;
	error_sys_log: DWORD;
	sys_time: TIME;
END_VAR
VAR // added by the converter: edge detectors and wires of the graphical bodies
    _w1, _w2 : ANY;
END_VAR

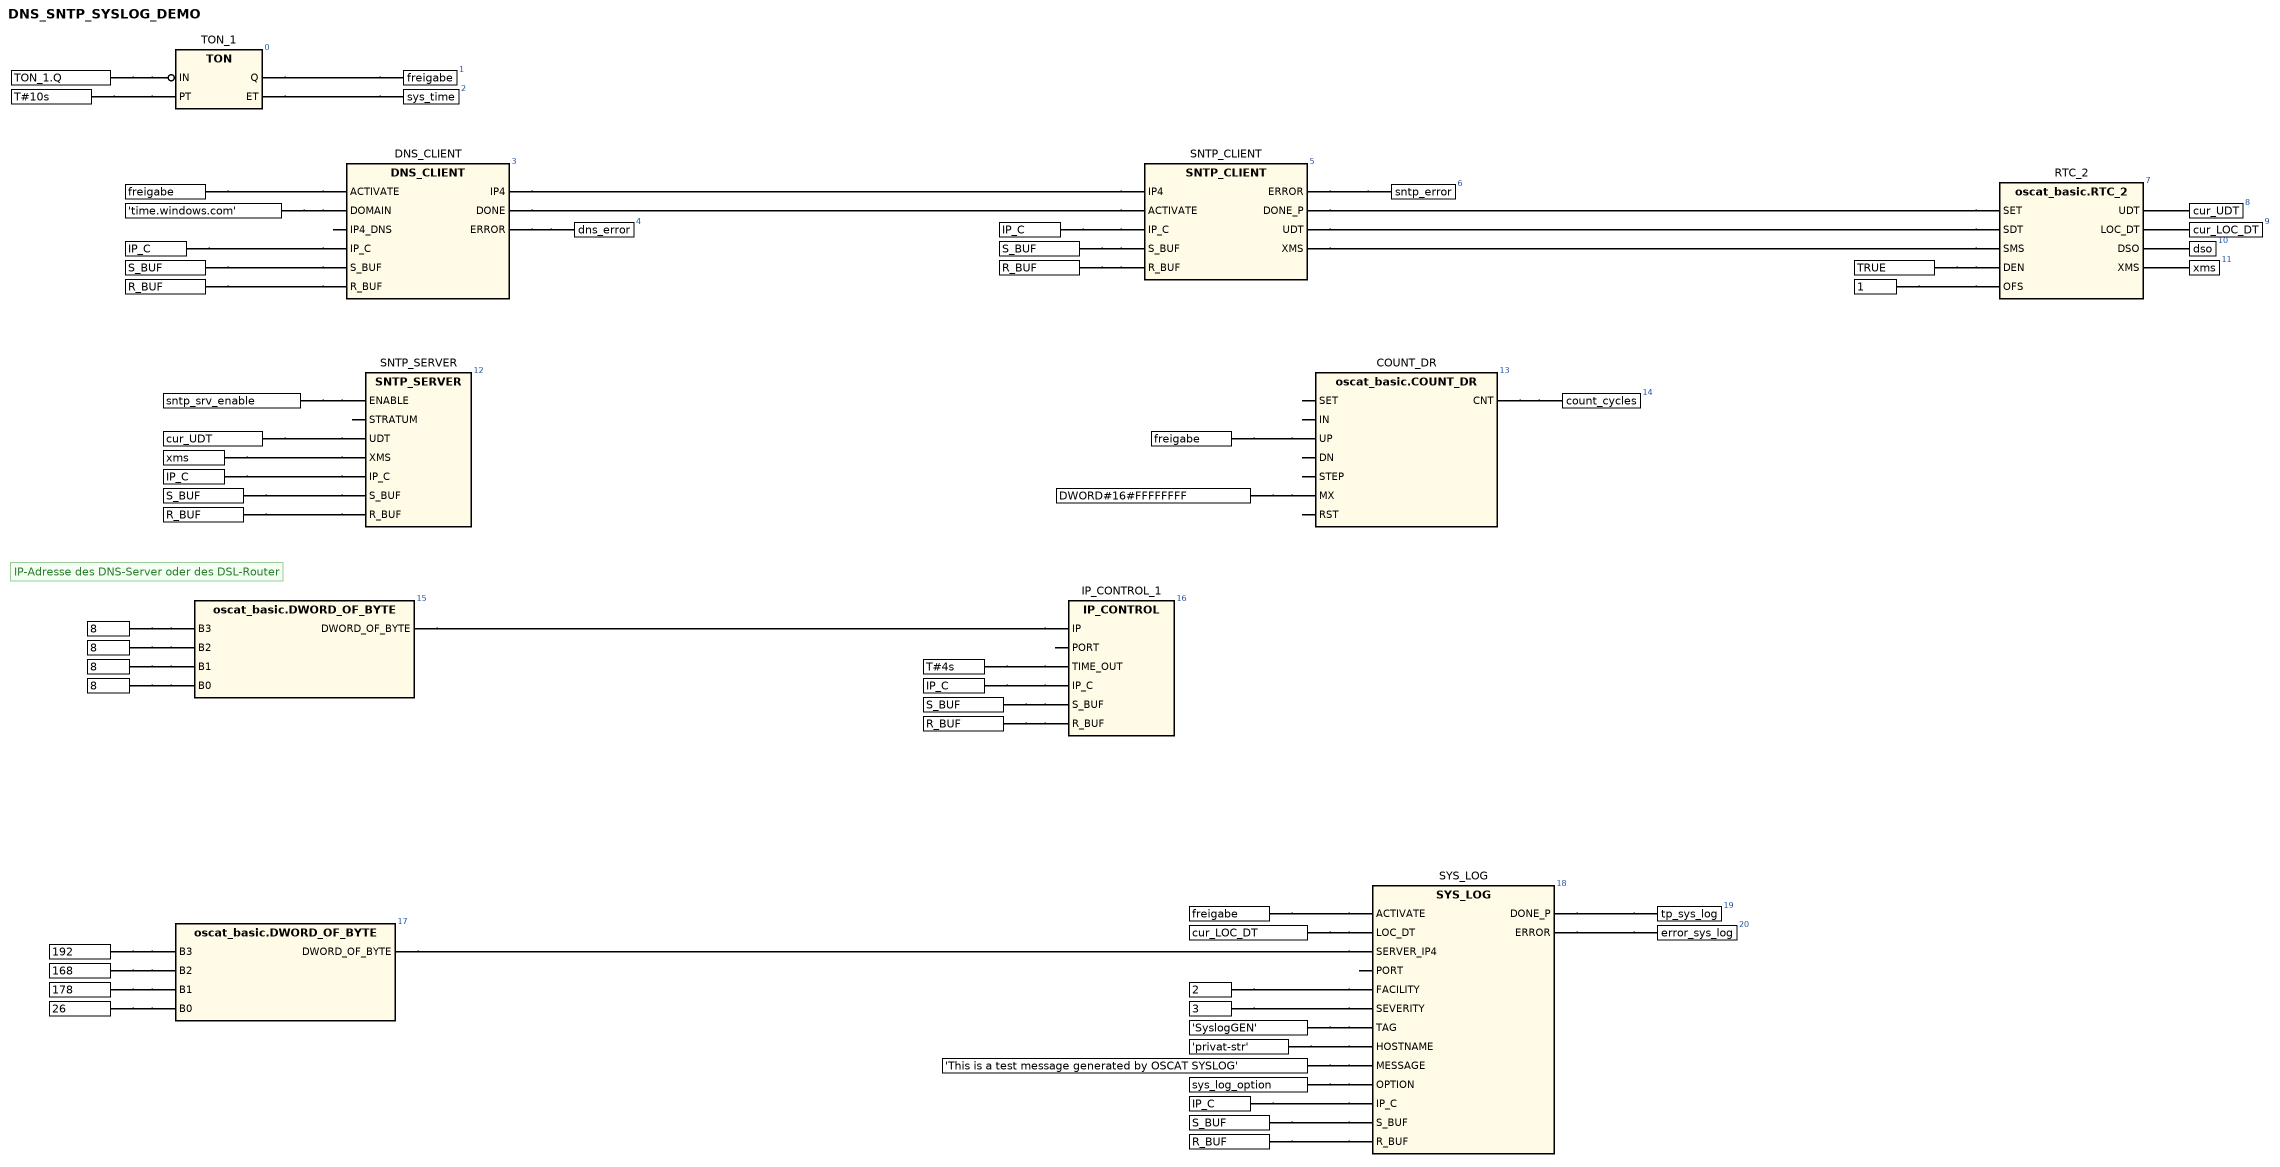
TON_1(IN := NOT TON_1.Q, PT := T#10s); // TON
freigabe := TON_1.Q;
sys_time := TON_1.ET;
DNS_CLIENT(ACTIVATE := freigabe, DOMAIN := 'time.windows.com', IP_C := IP_C, S_BUF := S_BUF, R_BUF := R_BUF);
dns_error := DNS_CLIENT.ERROR;
SNTP_CLIENT(IP4 := DNS_CLIENT.IP4, ACTIVATE := DNS_CLIENT.DONE, IP_C := IP_C, S_BUF := S_BUF, R_BUF := R_BUF);
sntp_error := SNTP_CLIENT.ERROR;
RTC_2(SET := SNTP_CLIENT.DONE_P, SDT := SNTP_CLIENT.UDT, SMS := SNTP_CLIENT.XMS, DEN := TRUE, OFS := 1); // oscat_basic.RTC_2
cur_UDT := RTC_2.UDT;
cur_LOC_DT := RTC_2.LOC_DT;
dso := RTC_2.DSO;
xms := RTC_2.XMS;
SNTP_SERVER(
    ENABLE := sntp_srv_enable,
    UDT := cur_UDT,
    XMS := xms,
    IP_C := IP_C,
    S_BUF := S_BUF,
    R_BUF := R_BUF);
COUNT_DR(UP := freigabe, MX := DWORD#16#FFFFFFFF); // oscat_basic.COUNT_DR
count_cycles := COUNT_DR.CNT;
// IP-Adresse des DNS-Server oder des DSL-Router
_w1 := oscat_basic.DWORD_OF_BYTE(B3 := 8, B2 := 8, B1 := 8, B0 := 8);
IP_CONTROL_1(IP := _w1, TIME_OUT := T#4s, IP_C := IP_C, S_BUF := S_BUF, R_BUF := R_BUF); // IP_CONTROL
_w2 := oscat_basic.DWORD_OF_BYTE(B3 := 192, B2 := 168, B1 := 178, B0 := 26);
SYS_LOG(
    ACTIVATE := freigabe,
    LOC_DT := cur_LOC_DT,
    SERVER_IP4 := _w2,
    FACILITY := 2,
    SEVERITY := 3,
    TAG := 'SyslogGEN',
    HOSTNAME := 'privat-str',
    MESSAGE := 'This is a test message generated by OSCAT SYSLOG',
    OPTION := sys_log_option,
    IP_C := IP_C,
    S_BUF := S_BUF,
    R_BUF := R_BUF);
tp_sys_log := SYS_LOG.DONE_P;
error_sys_log := SYS_LOG.ERROR;

END_PROGRAM

// POUs/NETWORK/SNTP_CLIENT
FUNCTION_BLOCK SNTP_CLIENT
VAR_IN_OUT
	IP_C : IP_C; (* IP_Control Verwaltungsstruktur *)
	S_BUF : NETWORK_BUFFER;
	R_BUF : NETWORK_BUFFER;
END_VAR
VAR_INPUT
	IP4 : DWORD;
	ACTIVATE : BOOL;
END_VAR
VAR_OUTPUT
	ERROR : DWORD;
	DONE_P : BOOL;
	UDT : DT;
	XMS : INT;
END_VAR
VAR
	IP_FIFO : IP_FIFO;
	ip_state : BYTE;
	ip_id : BYTE;
	i : INT;
	last : DWORD;
	state : INT;
	tx : DWORD;
	activate_last : BOOL;
	ip4_stored : DWORD;

	(*LOG_MSG : LOG_MSG;
	_debug_enable : BOOL := TRUE;*)

END_VAR

(*
version 1.1		20. oct. 2009
programmer 		ks
tested by		ks

SNTP_CLIENT führt eine SNTP-Anfrage bei einem SNTP/NTP-Server um die aktuelle Uhrzeit zu erhalten
*)

(* Domain Name System (query) *)
tx := OSCAT_BASIC.T_PLC_MS(); (* read system time *)

CASE state OF
00: (* auf positive Flanke SET warten *)
	DONE_P := FALSE;
	IF ACTIVATE AND NOT activate_last THEN
		ip4_stored := IP4; (* aktuelle IP4 speichern *)
		state := 10;
		ERROR := DWORD#0;
		ip_state := BYTE#1; (* Anmelden *)
		(*####################  DEBUG-MESSAGE  ###################################*)
		(*IF _debug_enable THEN
			LOG_CL.NEW_MSG := 'SNTP: S00 START';
			LOG_MSG();
		END_IF;*)
		(*########################################################################*)
	END_IF;

10: (* Bei IP_Control anmelden und auf freigabe warten *)
	IF ip_state = BYTE#3 THEN

		S_BUF.BUFFER[00] := BYTE#16#1B;
		FOR i := 1 TO 47 DO
			S_BUF.BUFFER[i] := BYTE#16#00;
		END_FOR;

		last := tx; (* aktuellen time wert sichern *)
		state := 30;

		(* IP Datenverkehr einrichten *)
		IP_C.C_PORT := WORD#123; (* Portnummer eintragen *)
		IP_C.C_IP := ip4_stored; (* IP eintragen *)
		IP_C.C_MODE := BYTE#1; (* Mode: UDP+AKTIV+PORT+IP *)
		IP_C.C_ENABLE := TRUE; (* Verbindungsaufbau freigeben *)
		IP_C.TIME_RESET := TRUE; (* Zeitueberwachung rücksetzen *)
		IP_C.R_OBSERVE := TRUE; (* Datenempfang ueberwachen *)
		S_BUF.SIZE := UINT#48; (* Sendelänge eintragen *)
		R_BUF.SIZE := UINT#0; (* Empfangslänge rücksetzen *)
    		(*####################  DEBUG-MESSAGE  ###################################*)
    		(*IF _debug_enable THEN
      			LOG_CL.NEW_MSG := 'SNTP: S10 SEND';
      			LOG_MSG();
    		END_IF;*)
    		(*########################################################################*)
	END_IF;

30:
	IF IP_C.ERROR <> DWORD#00 THEN
		ERROR := IP_C.ERROR;
		S_BUF.SIZE := UINT#0;
		R_BUF.SIZE := UINT#0;
		state := 0;
    		(*####################  DEBUG-MESSAGE  ###################################*)
    		(*IF _debug_enable THEN
      			LOG_CL.NEW_MSG := 'SNTP: S30 ERROR ~1';
      			LOG_CL.PRINTF[1] := DWORD_TO_STRING(ERROR);
      			LOG_MSG();
    		END_IF;*)
    		(*########################################################################*)

	ELSIF S_BUF.SIZE = UINT#0 AND R_BUF.SIZE >= UINT#48 THEN (* länge der empfangenen Daten prüfen *)

		(* Umrechnung SNTP Timestamp Base 1900-01-01 -> Unix 1970-01-01 = +2208988800 sekunden*)
		UDT := DWORD_TO_DT(OSCAT_BASIC.DWORD_OF_BYTE(R_BUF.BUFFER[40],R_BUF.BUFFER[41],R_BUF.BUFFER[42],R_BUF.BUFFER[43]) - DWORD#2208988800);

		(* Original-Sekundenanteile sind als 32 Bit Fractal dargestellt *)
		(* ms nur mit veringerte Auflösung berechnen 1/65535 -> Highword verwenden *)
		XMS := DWORD_TO_INT(SHR(DINT_TO_DWORD(WORD_TO_DINT(OSCAT_BASIC.WORD_OF_BYTE(R_BUF.BUFFER[44],R_BUF.BUFFER[45])) * DINT#1000),16));
		(* Zeitdifferenz (Laufzeitfehler) zwischen Send und Receive /2 teilen und addieren *)
		XMS := XMS + DWORD_TO_INT(SHR(tx - last,1));

		UDT := DWORD_TO_DT(DT_TO_DWORD(UDT) + (XMS / 1000)); (* sekundenanteile der Zeitdifferenz zu UDT aufrechnen *)
		XMS := XMS MOD 1000;  (* ms übernehmen *)
		state := 0;
		DONE_P := TRUE;
    		(*####################  DEBUG-MESSAGE  ###################################*)
    		(*IF _debug_enable THEN
        			LOG_CL.NEW_MSG := 'SNTP: S30 OK';
        			LOG_MSG();
    		END_IF;*)
    		(*########################################################################*)

	END_IF;

	IF state = 0 THEN
		IP_C.R_OBSERVE := FALSE; (* Datenempfang ueberwachen *)
		ip_state := BYTE#4;
	END_IF;

END_CASE;

activate_last := ACTIVATE; (* letzten Status sichern zur Flankenerkennung *)

(* IP_FIFO *)
IP_FIFO(FIFO:=IP_C.FIFO,STATE:=ip_state,ID:=ip_id);

(* revision history
ks	18. oct. 2008	rev 1.0
	original version

ks	20. oct. 2009	rev 1.1
	Networkbuffer und Buffer-funktionen auf Basis 0

*)

(***************************************************************************************)
(*               SNTP Datenstruktur
                                  1                   2                   3   
              0 1 2 3 4 5 6 7 8 9 0 1 2 3 4 5 6 7 8 9 0 1 2 3 4 5 6 7 8 9 0 1 
             +-+-+-+-+-+-+-+-+-+-+-+-+-+-+-+-+-+-+-+-+-+-+-+-+-+-+-+-+-+-+-+-+
Byte: 01-04  |LI | VN  |Mode |    Stratum    |     Poll      |   Precision   |
             +-+-+-+-+-+-+-+-+-+-+-+-+-+-+-+-+-+-+-+-+-+-+-+-+-+-+-+-+-+-+-+-+
Byte: 05-08  |                          Root  Delay (32 Bit)                 |
             +-+-+-+-+-+-+-+-+-+-+-+-+-+-+-+-+-+-+-+-+-+-+-+-+-+-+-+-+-+-+-+-+
Byte: 09-12  |                       Root  Dispersion (32 Bit)               |
             +-+-+-+-+-+-+-+-+-+-+-+-+-+-+-+-+-+-+-+-+-+-+-+-+-+-+-+-+-+-+-+-+
Byte: 13-16  |                     Reference Identifier (32 Bit)             |
             +-+-+-+-+-+-+-+-+-+-+-+-+-+-+-+-+-+-+-+-+-+-+-+-+-+-+-+-+-+-+-+-+
Byte: 17-24  |                    Reference Timestamp (64 Bit)               |
             +-+-+-+-+-+-+-+-+-+-+-+-+-+-+-+-+-+-+-+-+-+-+-+-+-+-+-+-+-+-+-+-+
Byte: 25-32  |                    Originate Timestamp (64 Bit)               |
             +-+-+-+-+-+-+-+-+-+-+-+-+-+-+-+-+-+-+-+-+-+-+-+-+-+-+-+-+-+-+-+-+
Byte: 33-40  |                     Receive Timestamp (64 Bit)                |
             +-+-+-+-+-+-+-+-+-+-+-+-+-+-+-+-+-+-+-+-+-+-+-+-+-+-+-+-+-+-+-+-+
Byte: 41-48  |                     Transmit Timestamp (64 Bit)               |
             +-+-+-+-+-+-+-+-+-+-+-+-+-+-+-+-+-+-+-+-+-+-+-+-+-+-+-+-+-+-+-+-+
Byte: 49-52  |                 Key Identifier (optional) (32 Bit)            |
             +-+-+-+-+-+-+-+-+-+-+-+-+-+-+-+-+-+-+-+-+-+-+-+-+-+-+-+-+-+-+-+-+
Byte: 53-68  |                 Message Digest (optional) (128 Bit)           |
             +-+-+-+-+-+-+-+-+-+-+-+-+-+-+-+-+-+-+-+-+-+-+-+-+-+-+-+-+-+-+-+-+

*)

(*
Worldwide NTP-Server


NIST-Zeitserver
• time-a.nist.gov
129.6.15.28 
NIST, Gaithersburg, Maryland 
• time-a.nist.gov
129.6.15.28 
NIST, Gaithersburg, Maryland 
• time-a.timefreq.bldrdoc.gov
132.163.4.101 (Stand: 1. Dezember 1999)
NIST, Boulder, Colorado 
• time-b.timefreq.bldrdoc.gov
132.163.4.102 (Stand: 1. Dezember 1999)
NIST, Boulder, Colorado 
• time-c.timefreq.bldrdoc.gov
132.163.4.103 (Stand: 1. Dezember 1999)
NIST, Boulder, Colorado 
• utcnist.colorado.edu
128.138.140.44
University of Colorado, Boulder 
• time.nist.gov
192.43.244.18
NCAR, Boulder, Colorado 
• time-nw.nist.gov
131.107.1.10
Microsoft, Redmond, Washington 
• nist1.dc.certifiedtime.com
216.200.93.8
Abovnet, North Virginia 
• nist1.datum.com
209.0.72.7
Datum, San Jose, Kalifornien 
• nist1.nyc.certifiedtime.com
208.184.49.129 
Abovnet, New York City 
• nist1.sjc.certifiedtime.com
207.126.103.202
Abovnet, San Jose, Kalifornien 

Zeitserver der ersten Ebene
Sortiert nach Standort: 
Nordamerika
• Palo Alto, Kalifornien: Systems Research Center, Compaq Computer Corp.
204.123.2.72: usno.pa-x.dec.com; CNAME: navobs1.pa-x.dec.com
Servicebereich: US-Zeitzonen PST (Pacific Standard Time) und MST (Mountain Standard Time) 
• Marina del Rey, Kalifornien: USC Information Sciences Institute
128.9.176.30: timekeeper.isi.edu
Servicebereich: CalRen2- und Los Nettos-Bereich  
• Washington, DC: U.S. Naval Observatory
192.5.41.41: tock.usno.navy.mil 
192.5.41.40: tick.usno.navy.mil
Servicebereich: NSFNET 
• Ottawa, Ontario, Kanada: National Research Council of Canada
time.chu.nrc.ca
Servicebereich: Kanada 
• Raleigh, North Carolina: North Carolina State University
152.1.58.124: terrapin.csc.ncsu.edu
Servicebereich: Südosten der USA 
• Cambridge, Massachusetts: MIT Information Systems
18.72.0.3: bitsy.mit.edu 
Servicebereich: NSFNET- und NEARnet-Bereich 
• Cambridge, Massachusetts: MIT
18.26.4.105: bonehed.lcs.mit.edu
Servicebereich: Osten der USA 
• Palo Alto, Kalifornien: Internet Software Consortium
192.5.5.250: clock.isc.org
Servicebereich: BARRnet, Alternet-West und CIX-West 
• Cambridge, Massachusetts: Open Software Foundation
130.105.4.59: clock.osf.org
Servicebereich: NSFNET- und NEARnet-Bereich 
• Palo Alto, Kalifornien: ViaNet Communications
209.81.9.7: clock.via.net 
• Cleveland, Ohio: Lewis Research Center (NASA)
128.156.1.43: lerc-dns.lerc.nasa.gov
Servicebereich: NSFNET und OARNET 
• Colorado Springs, Colorado: Schriever AFB
204.34.198.40: navobs1.usnogps.navy.mil; CNAME: tick.usnogps.navy.mil 
204.34.198.41: navobs1.usnogps.navy.mil; CNAME: tock.usnogps.navy.mil 
Servicebereich: US-Zeitzonen PST (Pacific Standard Time) und MST (Mountain Standard Time) 
• St. Louis, Missouri: Washington University
128.252.19.1: navobs1.usnogps.navy.mil; CNAME: tick.wustl.edu 
Servicebereich: US-Zeitzone CST (Central Standard Time) 
• Research Triangle Park, North Carolina: MCNC
192.101.21.1: ncnoc.ncren.net
Servicebereich: NC-REN-Bereich (North Carolina Research and Education Network) 
• Cupertino, Kalifornien: HP
192.6.38.127: ntp-cup.external.hp.com
Servicebereich: USA Westküste 
• Newark, Delaware: Conectiv Communications
138.39.7.20: ntp1.delmarva.com
Servicebereich: Cable & Wireless Network (früher MCInet) 
• University Park, Pennsylvania: Penn State University
128.118.46.3: otc1.psu.edu
Servicebereich: NSFNET, PREPNET und JvNCnet  

Europa
• Borowiec, Polen: Astrogeodynamical Observatory, Space Research Centre
150.254.183.15: vega.cbk.poznan.pl
Servicebereich: Polen und Europa 
• Stockholm, Schweden: Stupi AB
192.36.143.151: Time2.Stupi.SE
Servicebereich: Europa 
• Turin, Italien: IEN Galileo Ferraris
193.204.114.1: time.ien.it
Servicebereich: Italien und Europa 
• Zürich, Schweiz: Integrated Systems Laboratory , Eidgenössischen Technischen Hochschule Zürich 
129.132.2.21: swisstime.ethz.ch
Servicebereich: Schweiz und Europa 
• Turin, Italien: CSTV of National Research Council
150.145.33.1: tempo.cstv.to.cnr.it
Servicebereich: Italien und Europa 
• Erlangen, Deutschland: Universität Erlangen-Nürnberg
ntp0.fau.de; ntp1.fau.de; ntp2.fau.de; 
ntps1-0.uni-erlangen.de; ntps1-1.uni-erlangen.de; ntps1-2.uni-erlangen.de
Servicebereich: Deutschland und Europa 
• Berlin, Deutschland: Technische Universität Berlin
130.149.17.21: ntps1-0.cs.tu-berlin.de
130.149.17.8: ntps1-1.cs.tu-berlin.de
Servicebereich: Deutschland und Europa 
• Deutschland
131.173.17.7: ntps1-1.rz.Uni-Osnabrueck.DE
Servicebereich: Deutschland und Europa 
• Schweden
192.36.143.150: Time1.Stupi.SE
Servicebereich: SUnet und NORDUnet Schweden 

Fernost und pazifische Randgebiete
• Hong Kong: Chinesische Universität von Hong Kong. 
137.189.6.18: clock.cuhk.edu.hk
Servicebereich: Hong Kong (China) und Südostasien  
• Fukuoka, Japan: Universität Fukuoka
133.100.9.2: clock.nc.fukuoka-u.ac.jp
133.100.11.8: clock.tl.fukuoka-u.ac.jp
Servicebereich: Japan und pazifischer Raum  

Australien
• Melbourne, Australien: University of Melbourne
128.250.36.2: ntp.cs.mu.OZ.AU
Servicebereich: Australien und Neuseeland  

Zeitserver der zweiten Ebene
Nach geographischem Standort sortiert: 
Nordamerika
NTP-Zeitserver: • Quebec, Kanada: Canadian Meteorological Center
ntp1.cmc.ec.gc.ca; ntp2.cmc.ec.gc.ca 
Servicebereich: Ostkanada  
• Ontario, Kanada: National Research Council of Canada
time.chu.nrc.ca; time.nrc.ca
Servicebereich: Kanada 
• Saskatchewan, Kanada: University of Regina 
142.3.100.15: timelord.uregina.ca
Servicebereich: Kanada 
• Ontario, Kanada: University of Toronto
tick.utoronto.ca; tock.utoronto.ca
Servicebereich: Ostkanada  
• Mexiko: Audiotel-Büro 
ntp2a.audiotel.com.mx; ntp2c.audiotel.com.mx; ntp2b.audiotel.com.mx
Servicebereich: Avantel, MCINet und Mexiko 
• Santa Cruz, Kalifornien: Scruz-net, inc.
165.227.1.1: ns.scruz.net
Servicebereich: Westen der USA 
• San Diego, Kalifornien: UCSD Academic Computing Services/Network Operations
132.239.254.49: ntp.ucsd.edu
Servicebereich: CERFNET; NSFNET, SDSC-Bereich, und nahegelegene Bereiche 
• Quincy, Kalifornien 
ntp1.mainecoon.com; ntp2.mainecoon.com 
Servicebereich: Nordamerika 
• Newark, Delaware: University of Delaware
128.175.1.3: louie.udel.edu
Servicebereich: CAIRN, Abilene und vBNS  
• Atlanta, Georgia: CNSG
ntp.shorty.com
Servicebereich: Südwesten der USA  
• Kennesaw, Georgia: PeachNet 
rolex.peachnet.edu; timex.peachnet.edu
Servicebereich: PeachNet (Georgia) und Südwesten der USA  
• Urbana-Champaign, Illinois: University of Illinois
ntp-0.cso.uiuc.edu; ntp-1.cso.uiuc.edu; ntp-2.cso.uiuc.edu
Servicebereich: CICNET, Mittlerer Westen und NCSA-Bereich  
• Chicago, Illinois: Argonne National Laboratory 
ntp-1.mcs.anl.gov; ntp-2.mcs.anl.gov
Servicebereich: NSF/ANSNet, CICNet, NetIllinois und ESNet  
• West Lafayette, Indiana: Purdue University
gilbreth.ecn.purdue.edu; harbor.ecn.purdue.edu; molecule.ecn.purdue.edu 
Servicebereich: NSFNET- und CICNET-Bereich  
• Manhattan, Kansas: KansasNet OnLine Services
199.240.130.1: ntp1.kansas.net
199.240.130.12: ntp2.kansas.net
Servicebereich: Zentral-USA und Great Plains  
• Boston, Massachusetts: UMass-Boston CS dept.
158.121.104.4: timeserver.cs.umb.edu
Servicebereich: Neuengland  
• Minneapolis/St Paul, Minnesota: University of Minnesota
ns.nts.umn.edu; nss.nts.umn.edu
Servicebereich: CICNET-Bereich  
• Columbia, Missouri: University of Missouri-Columbia
128.206.206.12: everest.cclabs.missouri.edu
Servicebereich: MOREnet  
• Omaha, Nebraska: Radiks Internet Access
205.138.126.83: allison.radiks.net
Servicebereich: Mittlerer Westen, USA  
• Las Vegas, Nevada: University of Nevada System Computing Services
131.216.1.101: cuckoo.nevada.edu 
Servicebereich: NevadaNet, NSFNET und SDSC-Bereich  
• Las Vegas, Nevada: UNLV College of Engineering
tick.cs.unlv.edu; tock.cs.unlv.edu
Servicebereich: Sprintnet  
• New York City, New York: Columbia University
ntp.ctr.columbia.edu 
Servicebereich: Sprintlink und NYSERnet  
• Ithaca, New York: Cornell University 
192.35.82.50: ntp0.cornell.edu
Servicebereich: NSFNET und NYSER-Bereich  
• New York, New York: Morningside Campus, Columbia University
sundial.columbia.edu
Servicebereich: NYSERnet  
• New York City, New York: Columbia University Computer Science Department
timex.cs.columbia.edu 
Servicebereich: PSINET; NSFNET, und NYSER-Bereich  
• Norman, Oklahoma: University of Oklahoma
129.15.22.8: constellation.ecn.uoknor.edu 
Servicebereich: Midnet  
• Coos Bay, Oregon: Koala Computers
207.48.109.6: tick.koalas.com
Servicebereich: Nordwesten der USA  
• University Park, Pennsylvania: Penn State University
128.118.25.3: clock.psu.edu
Servicebereich: Internet2, vBNS, CERFnet(AT&T IP Services), PSC/NCNE und CASC 
• Pittsburgh, Pennsylvania: Pittsburgh Supercomputing Center
128.182.58.100: fuzz.psc.edu
Servicebereich: NSFNET und PSC-Bereich  
• Pittsburgh, Pennsylvania: Carnegie Mellon Electrical and Computer Engineering 
ntp-1.ece.cmu.edu; ntp-2.ece.cmu.edu 
Servicebereich: PREPNET und PSC-Bereich  
• Dallas, Texas: Cox School of Business, Southern Methodist University
129.119.80.126: ntp.cox.smu.edu 
Servicebereich: NSFNET und SESQUI-Bereich  
• Hughes Springs, Texas: First National Bank
209.144.20.76: ntp.fnbhs.com
Servicebereich: Nordosten Texas  
• Houston, Texas: Baylor College of Medicine
128.249.1.10: ntp.tmc.edu 
Servicebereich: NSFNET und SESQUI-Bereich  
• College Station, Texas: Texas A&M University
165.91.52.110: ntp5.tamu.edu
Servicebereich: NSFNET, SESQUI-Bereich, THEnet und TAMUSDSN 
• Plano, Texas: Greyware Automation Products
tick.greyware.com; tock.greyware.com
Servicebereich: Südzentral-USA  
• Blacksburg, Virginia: Virginia Tech Computing Center
ntp-1.vt.edu; ntp-2.vt.edu
Servicebereich: Südwesten der USA  
• Arlington, Virginia: Center for Seismic Studies
140.162.1.3: ntp.cmr.gov
Servicebereich: NSFNET und SURA-Bereich  
• Richland, Washington: Washington State University 
192.31.216.30: clock.tricity.wsu.edu
Servicebereich: NSFNET und NorthWestNet  
• Washington, USA: Mill Creek
time.ultimeth.net
Servicebereich: Nordwesten der USA  
• Wisconsin, USA: Computer Science Department, University of Wisconsin-Madison
ntp1.cs.wisc.edu; ntp2.cs.wisc.edu; ntp3.cs.wisc.edu
Servicebereich: USA und jeder andere  

Südamerika
• Buenos Aires, Argentinien: Network Access Point
200.49.40.1: CNAME: tick.nap.com.ar
200.49.32.1: CNAME: tock.nap.com.ar
Servicebereich: Argentinien 
• Buenos Aires, Argentinien: Sinectis S.A.
time.sinectis.com.ar 
Servicebereich: Argentinien 
• Brasilien: Brazilian Research Network
200.144.121.33: ntp.cais.rnp.br 
Servicebereich: Brasilien 
• Venezuela: VELUG, Grupo de Usuarios Linux de Venezuela
150.185.192.250: ntp.linux.org.ve
Servicebereich: Arica  

Europa
• Zürich, Schweiz: Eidgenössischen Technischen Hochschule Zürich
129.132.98.11: bernina.ethz.ch
Servicebereich: Schweiz und Europa  
• Standort: Kopenhagen, Dänemark, Europa 
clock.netcetera.dk; clock2.netcetera.dk 
Servicebereich: Dänemark, Skandinavien und Nordeuropa  
• Spanien: Altea 
slug.ctv.es
Servicebereich: Spanien  
• Pieksamaki, Finnland: Keski-Savon Oppimiskeskus
tick.keso.fi; tock.keso.fi
Servicebereich: Finnland  
• Meudon, Frankreich: Observatoire de Paris-Meudon 
ntp.obspm.fr 
Servicebereich: Frankreich und Europa  
• Lyon, Frankreich: CISM 
ntp.univ-lyon1.fr 
Servicebereich: Frankreich, Schweiz, Italien und Europa  
• Paris, Frankreich: VIA, Ecole Centrale
138.195.130.70: ntp.via.ecp.fr
Servicebereich: Frankreich und Europa  
• Budapest, Ungarn: KFKI Research Institute for Particle and Nuclear Physics
148.6.0.1: time.kfki.hu
Servicebereich: HUNGARNET  
• Italien: Net4u Srl, Vercelli, Italien
195.32.52.129: ntps.net4u.it
Servicebereich: Italien  
• Oslo, Norwegen: Universität Oslo
129.240.64.3: fartein.ifi.uio.no 
Servicebereich: NORDUnet  
• Oslo, Norwegen: Alcanet International
time.alcanet.no
Servicebereich: Europa 
• Krakau, Polen: Academic Computer Centre 
149.156.4.11: info.cyf-kr.edu.pl
Servicebereich: Polen und Europa  
• Lund, Schweden: Lund Institute of Technology
130.235.20.3: ntp.lth.se 
Servicebereich: Schweden und NORDUnet 
• Ljubljana, Slowenien: Institute of Biophysics, University of Ljubljana
biofiz.mf.uni-lj.si 193.2.69.11
Servicebereich: Slowenien und Europa  
• Ljubljana, Slowenien: Hydrometeorological Institute of Slovenia
hmljhp.rzs-hm.si
Servicebereich: Slowenien und Europa  
• Ljubljana, Slowenien: Academic and Research Network of Slovenia
ntp1.arnes.si; ntp2.arnes.si
Servicebereich: Slowenien und Europa  
• Ljubljana, Slowenien: J. Stefan Institute
time.ijs.si
Servicebereich: Slowenien und Europa  

Britische Inseln
• Dublin, Irland: School of Mathematics, Trinity College 
ntp.cs.tcd.ie; ntp.maths.tcd.ie; ntp.tcd.ie
Servicebereich: Irland und Großbritannien 
• Glasgow, Schottland: Strathclyde University 
ntp.cs.strath.ac.uk 
Servicebereich: Großbritannien, Europa und andere 
• Cambridge, Großbritannien
ntp0.uk.uu.net; ntp1.uk.uu.net; 
ntp2.uk.uu.net 
Servicebereich: UUNET (in Großbritannien früher auch als PIPEX bekannt) und Großbritannien.  
• Manchester, England: University of Manchester
ntp2a.mcc.ac.uk; ntp2b.mcc.ac.uk;
ntp2c.mcc.ac.uk; ntp2d.mcc.ac.uk 
Servicebereich: Großbritannien  
• Buckinghamshire, Großbritannien: Wibble U.K., Aylesbury
tick.tanac.net
Servicebereich: Großbritannien  

Asien
• Moskau, Russland: Landau Institute for Theoretical Physics
193.233.9.7: ntp.landau.ac.ru
Servicebereich: Russland  
• Russland: Pushchino (bei Moskau)
194.149.67.130: ntp.psn.ru
Servicebereich: Russland 
• Chernogolovka, Russland: Chernogolovka Scientific Center (bei Moskau)
193.233.46.10: sign.chg.ru
Servicebereich: Russland  

Fernost und pazifische Randgebiete
• Tokyo, Japan: Cyber Fleet, Inc.
203.139.30.195: ntp.cyber-fleet.net
Servicebereich: Japan und Ostasien  
• Seoul, Korea: Inet, Inc.
time.nuri.net
Servicebereich: Korea, Japan, Hong Kong und Ostasien  
• Hamilton, Neuseeland: Universität Waikato
truechimer.waikato.ac.nz; truechimer1.waikato.ac.nz; 
truechimer2.waikato.ac.nz; truechimer3.waikato.ac.nz
Servicebereich: Neuseeland  
• Singapur und Philippinen: 
ntp.shim.org 
Servicebereich: Singapur  

Afrika
• Lagos, Nigeria: Supernet300
ntp.supernet300.com
Servicebereich: Westafrika (hauptsächlich nigerischer NITEL-Backbone)  
• Pietermaritzburg, Südafrika: Natal University
143.128.82.200: ntp.cs.unp.ac.za
Servicebereich: Südafrika  

Australien
• Adelaide, Südaustralien: University of Adelaide
129.127.28.4: augean.eleceng.adelaide.edu.au
129.127.40.3: ntp.adelaide.edu.au
203.21.37.18: ntp.saard.net
Servicebereich: AARNet  
• Carlton, Victoria, Australien: eSec Limited
203.21.84.4: time.esec.com.au  

*)

END_FUNCTION_BLOCK

// POUs/NETWORK/SNTP_SERVER
FUNCTION_BLOCK SNTP_SERVER
VAR_IN_OUT
	IP_C : IP_C; (* IP_Control Verwaltungsstruktur *)
	S_BUF : NETWORK_BUFFER;
	R_BUF : NETWORK_BUFFER;
END_VAR
VAR_INPUT
	ENABLE : BOOL;
	STRATUM : BYTE := BYTE#1;
	UDT : DT;
	XMS : INT;
END_VAR
VAR
	IP_FIFO : IP_FIFO;
	ip_state : BYTE;
	ip_id : BYTE;
	i2 : INT;
	i : INT;
	timestamp_int : DWORD; (* Timestamp integer part *)
	timestamp_sek : DWORD; (* Timestamp fraction part (HIGH_WORD) *)
	ts_b : BYTE;
	state : INT;
	tx : UDINT;
	t : TON;

	(*LOG_MSG : LOG_MSG;
	_debug_enable : BOOL := TRUE;*)

END_VAR

(*
version 1.2		17. may. 2011
programmer 		ks
tested by			ks

SNTP_SERVER stellt Datum/Uhrzeit füR andere (S)NTP_CLIENTS zur Verfügung.
*)

(* Domain Name System (query) *)
tx := OSCAT_BASIC.T_PLC_MS(); (* read system time *)

CASE state OF

00: (* Warten auf Freigabe *)
	IF ENABLE THEN
		state := 10;
		ip_state := BYTE#1; (* Anmelden *)
    		(*####################  DEBUG-MESSAGE  ###################################*)
    		(*IF _debug_enable THEN
      			LOG_CL.NEW_MSG := 'SNTP_SERVER: S00 START';
      			LOG_MSG();
    		END_IF;*)
    		(*########################################################################*)
	END_IF;

10: (* Bei IP_Control anmelden und auf freigabe warten *)
	IF ip_state = BYTE#3 THEN
		(* IP Datenverkehr einrichten *)
		IP_C.C_PORT := WORD#123; (* Portnummer eintragen *)
		IP_C.C_IP := DWORD#00; (* IP eintragen *)
		IP_C.C_MODE := BYTE#5; (* Mode: UDP+PASSIV+PORT *)
		IP_C.C_ENABLE := TRUE; (* Verbindungsaufbau freigeben *)
		IP_C.TIME_RESET := TRUE; (* Zeitueberwachung rücksetzen *)
		IP_C.R_OBSERVE := FALSE; (* Datenempfang ueberwachen *)
		S_BUF.SIZE := UINT#0; (* Sendelänge eintragen *)
		R_BUF.SIZE := UINT#0; (* Empfangslänge rücksetzen *)
		state := 20;
    		(*####################  DEBUG-MESSAGE  ###################################*)
    		(*IF _debug_enable THEN
      			LOG_CL.NEW_MSG := 'SNTP_SERVER: S10 INIT';
      			LOG_MSG();
    		END_IF;*)
    		(*########################################################################*)
	END_IF;
20:
	IF R_BUF.SIZE > UINT#0 THEN
		state := 20;
    		(*####################  DEBUG-MESSAGE  ###################################*)
    		(*IF _debug_enable THEN
      			LOG_CL.NEW_MSG := 'SNTP_SERVER: S20 REQUEST - Size: ~1';
      			LOG_CL.PRINTF[1] := UINT_TO_STRING(R_BUF.SIZE);
      			LOG_MSG();
    		END_IF;*)
    		(*########################################################################*)
		(* empfangenes Telegramm mit 00 auffüllen , wenn zu kurz ! und Sendebuffer mit 00 vorbelegen *)
		FOR i := 0 TO 47 DO
			IF INT_TO_UINT(i) > R_BUF.SIZE - 1 THEN
				R_BUF.BUFFER[i] := BYTE#00;
			END_IF;
			S_BUF.BUFFER[i] := BYTE#00;
		END_FOR;

		R_BUF.SIZE := UINT#0;

		(* Sendedaten aufbereiten *)
		S_BUF.BUFFER[0] := BYTE#2#11100; (* Flags: NO WARNING, NTP VERSION 3 , SERVER *)
		S_BUF.BUFFER[1] := STRATUM; (* Peer Clock Stratum: *)
		S_BUF.BUFFER[2] := BYTE#10; (* Peer Polling Intervall 2 hoch 10 = 1024 sek. *)
		S_BUF.BUFFER[3] := BYTE#16#FB; (* Peer Clock Precision: -5 = -31,25ms *)

		(* Umrechnung SNTP Timestamp Base 1900-01-01 = Unix 1970-01-01 + 2208988800 sekunden *)
		timestamp_int := DT_TO_DWORD(UDT) + DWORD#2208988800;

		(* Sekundenanteile sind als 32 Bit Fractal dargestellt *)
		(* nur mit veringerte Auflösung berechnen 1/65535 -> Highword verwenden *)
		(* Berechnung des Sekundenanteils: xms * 65535 / 1000 *)
		timestamp_sek := DINT_TO_DWORD(DWORD_TO_DINT(SHL(INT_TO_DWORD(XMS),16))/DINT#1000);

		ts_b := OSCAT_BASIC.BYTE_OF_DWORD(timestamp_int,3); (* Timestamp Byte 3 *)
		S_BUF.BUFFER[16] := ts_b; (* Reference Timestamp *)
		S_BUF.BUFFER[32] := ts_b; (* Receive   Timestamp *)
		S_BUF.BUFFER[40] := ts_b; (* Transmit  Timestamp *)

		ts_b := OSCAT_BASIC.BYTE_OF_DWORD(TIMESTAMP_INT,2); (* Timestamp Byte 2 *)
		S_BUF.BUFFER[17] := ts_b; (* Reference Timestamp *)
		S_BUF.BUFFER[33] := ts_b; (* Receive   Timestamp *)
		S_BUF.BUFFER[41] := ts_b; (* Transmit  Timestamp *)

		ts_b := OSCAT_BASIC.BYTE_OF_DWORD(TIMESTAMP_INT,1); (* Timestamp Byte 1 *)
		S_BUF.BUFFER[18] := ts_b; (* Reference Timestamp *)
		S_BUF.BUFFER[34] := ts_b; (* Receive   Timestamp *)
		S_BUF.BUFFER[42] := ts_b; (* Transmit  Timestamp *)

		ts_b := OSCAT_BASIC.BYTE_OF_DWORD(TIMESTAMP_INT,0); (* Timestamp Byte 0 *)
		S_BUF.BUFFER[19] := ts_b; (* Reference Timestamp *)
		S_BUF.BUFFER[35] := ts_b; (* Receive   Timestamp *)
		S_BUF.BUFFER[43] := ts_b; (* Transmit  Timestamp *)

		ts_b := OSCAT_BASIC.BYTE_OF_DWORD(TIMESTAMP_SEK,1); (* Timestamp Byte 1 *)
		S_BUF.BUFFER[20] := ts_b; (* Reference Timestamp *)
		S_BUF.BUFFER[36] := ts_b; (* Receive   Timestamp *)
		S_BUF.BUFFER[44] := ts_b; (* Transmit  Timestamp *)

		ts_b := OSCAT_BASIC.BYTE_OF_DWORD(timestamp_sek,0);	(* Timestamp Byte 0 *)
		S_BUF.BUFFER[21] := ts_b; (* Reference Timestamp *)
		S_BUF.BUFFER[37] := ts_b; (* Receive   Timestamp *)
		S_BUF.BUFFER[45] := ts_b; (* Transmit  Timestamp *)

		(* Byte 1-8 von Transmit-Time auf Originate-Time umkopieren *)
		i2 := 40;
		FOR i := 24 TO 31 DO
			S_BUF.BUFFER[i] := R_BUF.BUFFER[i2];
			i2 := i2 +1;
		END_FOR;

		S_BUF.SIZE := UINT#48; (* Daten senden *)

	ELSIF NOT ENABLE AND S_BUF.SIZE = UINT#0 THEN
		ip_state := BYTE#4; (* Abmelden *)
		state := 0;
	END_IF;

END_CASE;

t(IN:= IP_C.ERROR > DWORD#0, PT:=T#5s);
IF t.Q THEN
  IP_C.TIME_RESET := TRUE; (* Error Reset *)
END_IF;

(* IP_FIFO *)
IP_FIFO(FIFO:=IP_C.FIFO,STATE:=ip_state,ID:=ip_id);

(* revision history
ks	18. oct. 2008	rev 1.0
	original version

ks	20. oct. 2009	rev 1.1
	Networkbuffer und Buffer-funktionen auf Basis 0

ks	17. may. 2011	rev 1.2
	automatischer re-connect
*)


(*               SNTP(NTP) Datenstruktur
                                  1                   2                   3
              0 1 2 3 4 5 6 7 8 9 0 1 2 3 4 5 6 7 8 9 0 1 2 3 4 5 6 7 8 9 0 1
             +-+-+-+-+-+-+-+-+-+-+-+-+-+-+-+-+-+-+-+-+-+-+-+-+-+-+-+-+-+-+-+-+
Byte: 01-04  |LI | VN  |Mode |    Stratum    |     Poll      |   Precision   |
             +-+-+-+-+-+-+-+-+-+-+-+-+-+-+-+-+-+-+-+-+-+-+-+-+-+-+-+-+-+-+-+-+
Byte: 05-08  |                          Root  Delay (32 Bit)                 |
             +-+-+-+-+-+-+-+-+-+-+-+-+-+-+-+-+-+-+-+-+-+-+-+-+-+-+-+-+-+-+-+-+
Byte: 09-12  |                       Root  Dispersion (32 Bit)               |
             +-+-+-+-+-+-+-+-+-+-+-+-+-+-+-+-+-+-+-+-+-+-+-+-+-+-+-+-+-+-+-+-+
Byte: 13-16  |                     Reference Identifier (32 Bit)             |
             +-+-+-+-+-+-+-+-+-+-+-+-+-+-+-+-+-+-+-+-+-+-+-+-+-+-+-+-+-+-+-+-+
Byte: 17-24  |                    Reference Timestamp (64 Bit)               |
             +-+-+-+-+-+-+-+-+-+-+-+-+-+-+-+-+-+-+-+-+-+-+-+-+-+-+-+-+-+-+-+-+
Byte: 25-32  |                    Originate Timestamp (64 Bit)               |
             +-+-+-+-+-+-+-+-+-+-+-+-+-+-+-+-+-+-+-+-+-+-+-+-+-+-+-+-+-+-+-+-+
Byte: 33-40  |                     Receive Timestamp (64 Bit)                |
             +-+-+-+-+-+-+-+-+-+-+-+-+-+-+-+-+-+-+-+-+-+-+-+-+-+-+-+-+-+-+-+-+
Byte: 41-48  |                     Transmit Timestamp (64 Bit)               |
             +-+-+-+-+-+-+-+-+-+-+-+-+-+-+-+-+-+-+-+-+-+-+-+-+-+-+-+-+-+-+-+-+
Byte: 49-52  |                 Key Identifier (optional) (32 Bit)            |
             +-+-+-+-+-+-+-+-+-+-+-+-+-+-+-+-+-+-+-+-+-+-+-+-+-+-+-+-+-+-+-+-+
Byte: 53-68  |                 Message Digest (optional) (128 Bit)           |
             +-+-+-+-+-+-+-+-+-+-+-+-+-+-+-+-+-+-+-+-+-+-+-+-+-+-+-+-+-+-+-+-+
*)

END_FUNCTION_BLOCK

// POUs/NETWORK/SYS_LOG
FUNCTION_BLOCK SYS_LOG
VAR_IN_OUT
	IP_C : IP_C; (* IP_Control Verwaltungsstruktur *)
	S_BUF : NETWORK_BUFFER;
	R_BUF : NETWORK_BUFFER;
END_VAR
VAR_INPUT
	ACTIVATE : BOOL;
	LOC_DT : DT;
	SERVER_IP4 : DWORD;
	PORT : WORD;
	FACILITY : BYTE;
	SEVERITY : BYTE;
	TAG : STRING(32);
	HOSTNAME : STRING;
	MESSAGE : STRING(OSCAT_BASIC.STRING_LENGTH);
	OPTION : BYTE;
END_VAR
VAR_OUTPUT
	DONE_P : BOOL;
	ERROR : DWORD;
END_VAR
VAR
	ip_state : BYTE;
	ip_id : BYTE;
	IP_FIFO : IP_FIFO;
	activate_last : BOOL;
	state : INT;
	s1 : STRING(20);
	i : INT;

	(*LOG_MSG : LOG_MSG;
	_debug_enable : BOOL := TRUE;*)

END_VAR

(*
version 1.1		20. jun. 2009
programmer 		ks
tested by		ks

SYSLOG versendet Meldungen auf Basis des SYSLOG-Standards

*)

CASE state OF
00: (* auf positive Flanke SET warten *)
	IF ACTIVATE AND NOT ACTIVATE_LAST THEN
		state := 10;
		ERROR := DWORD#0;
		IP_STATE := BYTE#1; (* Anmelden *)
    		(*####################  DEBUG-MESSAGE  ###################################*)
    		(*IF _debug_enable THEN
      			LOG_CL.NEW_MSG := 'SYS_LOG: S00 START /IP_ID ~4';
      			LOG_CL.PRINTF[4]  := BYTE_TO_STRING(IP_ID);
      			LOG_MSG();
    		END_IF;*)
    		(*########################################################################*)
	END_IF;
	DONE_P := FALSE;

10: (* Bei IP_Control anmelden und auf freigabe warten *)
	IF IP_STATE = BYTE#3 THEN
		(* Sendedaten aufbereiten *)
		i := 0;
		IF (OPTION AND BYTE#0000_0001) = BYTE#00 THEN (* Option: no priority Code *)
			(* Priority:  '<xx>' als dezimalwert *)
			(* BYTE: xxxx x...  = Facility *)
			(*       .... .xxx  = Level *)
			s1 := REPLACE('<P>',BYTE_TO_STRING(SHL(FACILITY,3) OR (SEVERITY AND BYTE#0000_0111)),1,2);
		ELSE
			s1 := '';
		END_IF;

		IF (OPTION AND BYTE#0000_0010) = BYTE#00 THEN (* Option: No Use Syslog RFC Header *)
			(* 'month day hh:mm:ss ' *)
			s1 := CONCAT(s1,OSCAT_BASIC.DT_TO_STRF(DTI:=LOC_DT,MS:=0,FMT:='#E #W #N:#R:#T ',LANG:=1));
			OSCAT_BASIC._STRING_TO_BUFFER(STR:=s1,POS:=i,PT:=ADR(S_BUF.BUFFER),SIZE:=UINT#1024);
			i := i + LEN(s1);
			(* ' sourcename eintragen *)
			OSCAT_BASIC._STRING_TO_BUFFER(STR:=HOSTNAME,POS:=i,PT:=ADR(S_BUF.BUFFER),SIZE:=UINT#1024);
			i := i + LEN(HOSTNAME);
			S_BUF.BUFFER[i] := BYTE#32; (* leerzeichen einfuegen *)
			i := i + 1;
			(* ' tag eintragen *)
			OSCAT_BASIC._STRING_TO_BUFFER(STR:=TAG,POS:=i,PT:=ADR(S_BUF.BUFFER),SIZE:=UINT#1024);
			i := i + LEN(TAG);
			S_BUF.BUFFER[i] := BYTE#32; (* leerzeichen einfuegen *)
			i := i + 1;
		END_IF;

		(* ' message eintragen *)
		OSCAT_BASIC._STRING_TO_BUFFER(STR:=MESSAGE,POS:=i,PT:=ADR(S_BUF.BUFFER),SIZE:=UINT#1024);
		i := i + LEN(MESSAGE);

		IF (OPTION AND BYTE#0000_0100) > BYTE#00 THEN (* Option: Add a CR & LF to end of message *)
			S_BUF.BUFFER[i] := BYTE#13; (* Carriage Return einfuegen *)
			i := i + 1;
			S_BUF.BUFFER[i] := BYTE#10; (* Linefeed einfuegen *)
			i := i + 1;
		END_IF;

		state := 30;

		(* IP Datenverkehr einrichten *)
		IF (OPTION AND BYTE#2#0000_1000) > BYTE#00 THEN (* Option: TCP Mode *)
			IP_C.C_MODE := BYTE#0; (* Mode: TCP/AKTIV *)
		ELSE
			IP_C.C_MODE := BYTE#1; (* Mode: UDP/AKTIV *)
		END_IF;

		IF PORT = WORD#0 THEN (* keine Portnummer vorgegeben ? *)
			IF IP_C.C_MODE = BYTE#0 THEN (* Modus bestimmen  TCP oder UDP ? *)
				IP_C.C_PORT := WORD#1468; (* Standard Portnummer für Syslog over TCP *)
			ELSE
				IP_C.C_PORT := WORD#514; (* Standard Portnummer für Syslog over UDP *)
			END_IF;
		ELSE
			IP_C.C_PORT := PORT; (* uebergebene Portnummer eintragen *)
		END_IF;

		IP_C.C_IP := SERVER_IP4; (* IP eintragen *)
		IP_C.C_ENABLE := TRUE; (* Verbindungsaufbau freigeben *)
		IP_C.TIME_RESET := TRUE; (* Zeitueberwachung rücksetzen *)
		IP_C.R_OBSERVE := FALSE; (* Datenempfang ueberwachen *)
		S_BUF.SIZE := INT_TO_UINT(i); (* Sendelänge eintragen *)
		R_BUF.SIZE := UINT#0; (* Empfangslänge rücksetzen *)
    		(*####################  DEBUG-MESSAGE  ###################################*)
    		(*IF _debug_enable THEN
      			LOG_CL.NEW_MSG := 'SYS_LOG: S20 SEND /IP_ID ~4';
      			LOG_CL.PRINTF[4]  := BYTE_TO_STRING(IP_ID);
      			LOG_MSG();
    		END_IF;*)
    		(*########################################################################*)
	END_IF;

30:
	IF IP_C.ERROR <> DWORD#00 THEN
		ERROR := IP_C.ERROR;
		state := 0;
    		(*####################  DEBUG-MESSAGE  ###################################*)
    		(*IF _debug_enable THEN
      			LOG_CL.NEW_MSG := 'SYS_LOG: S30 ERROR ~1 IP_ID ~4';
      			LOG_CL.PRINTF[1]  := DWORD_TO_STRING(ERROR);
      			LOG_CL.PRINTF[4]  := BYTE_TO_STRING(IP_ID);
      			LOG_MSG();
    		END_IF;*)
    		(*########################################################################*)
	ELSIF S_BUF.SIZE = UINT#0 THEN (* warten bis alle daten gesendet sind *)
		DONE_P := TRUE;
		state := 0;
    		(*####################  DEBUG-MESSAGE  ###################################*)
    		(*IF _debug_enable THEN
      			LOG_CL.NEW_MSG := 'SYS_LOG: S30 OK /IP_ID ~4';
      			LOG_CL.PRINTF[4]  := BYTE_TO_STRING(IP_ID);
      			LOG_MSG();
    		END_IF;*)
    		(*########################################################################*)
	END_IF;

	IF state = 0 THEN (* Verbindung freigeben *)
		IP_STATE := BYTE#4;
	END_IF;

END_CASE;

ACTIVATE_LAST := ACTIVATE; (* letzten Status sichern zur Flankenerkennung *)

(* IP_FIFO *)
IP_FIFO(FIFO:=IP_C.FIFO,STATE:=ip_state,ID:=IP_ID);

(* revision history
ks	18. oct. 2008	rev 1.0
	original version

ks	20. jun. 2009	rev 1.1
	Networkbuffer und Buffer-funktionen auf Basis 0

*)

END_FUNCTION_BLOCK

// POUs/DEMO/FILE_BLOCK_DEMO
PROGRAM FILE_BLOCK_DEMO
VAR
	PT : NETWORK_BUFFER;
	fsd : FILE_SERVER_DATA;
	FILE_SERVER : FILE_SERVER;
	FILE_BLOCK : FILE_BLOCK;
	filename : STRING := 'config.ini';
	data : BYTE;
	error : BYTE;
	mode : BYTE;
	pos : UDINT;
END_VAR

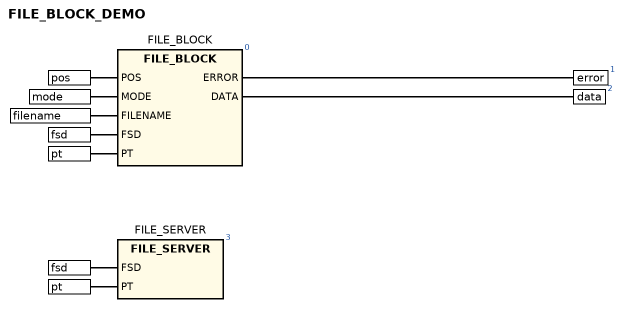
FILE_BLOCK(POS := pos, MODE := mode, FILENAME := filename, FSD := fsd, PT := pt);
error := FILE_BLOCK.ERROR;
data := FILE_BLOCK.DATA;
FILE_SERVER(FSD := fsd, PT := pt);

END_PROGRAM

// POUs/DEMO/FTP_CLIENT_DEMO
PROGRAM FTP_CLIENT_DEMO
VAR
	FTP_CLIENT: FTP_CLIENT;
	ftp_activate: BOOL;
	ftp_done: BOOL;
	ftp_busy: BOOL;
	ftp_error_c: DWORD;
	ftp_error_t: BYTE;
	ftp_url: STRING := 'ftp://581920:123456@oscat.atwebpages.com:2000/subordner/';
	ftp_filename: STRING := '0100kb.bin';
	ftp_download: BOOL := TRUE;
	ftp_activ: BOOL := FALSE;
	file_delete: BOOL := FALSE;
	ftp_timeout: TIME := T#30s;
	zeit : TIME := T#30s;
	stop: BOOL;
	start: BOOL :=TRUE ;
	reset: BOOL;
	error: DWORD;
	ok: DWORD;
	CLK_PRG_1: oscat_basic.CLK_PRG;
	COUNT_DR_1: oscat_basic.COUNT_DR;
	COUNT_DR_2: oscat_basic.COUNT_DR;
END_VAR
VAR // added by the converter: edge detectors and wires of the graphical bodies
    _w1, _w2 : ANY;
END_VAR

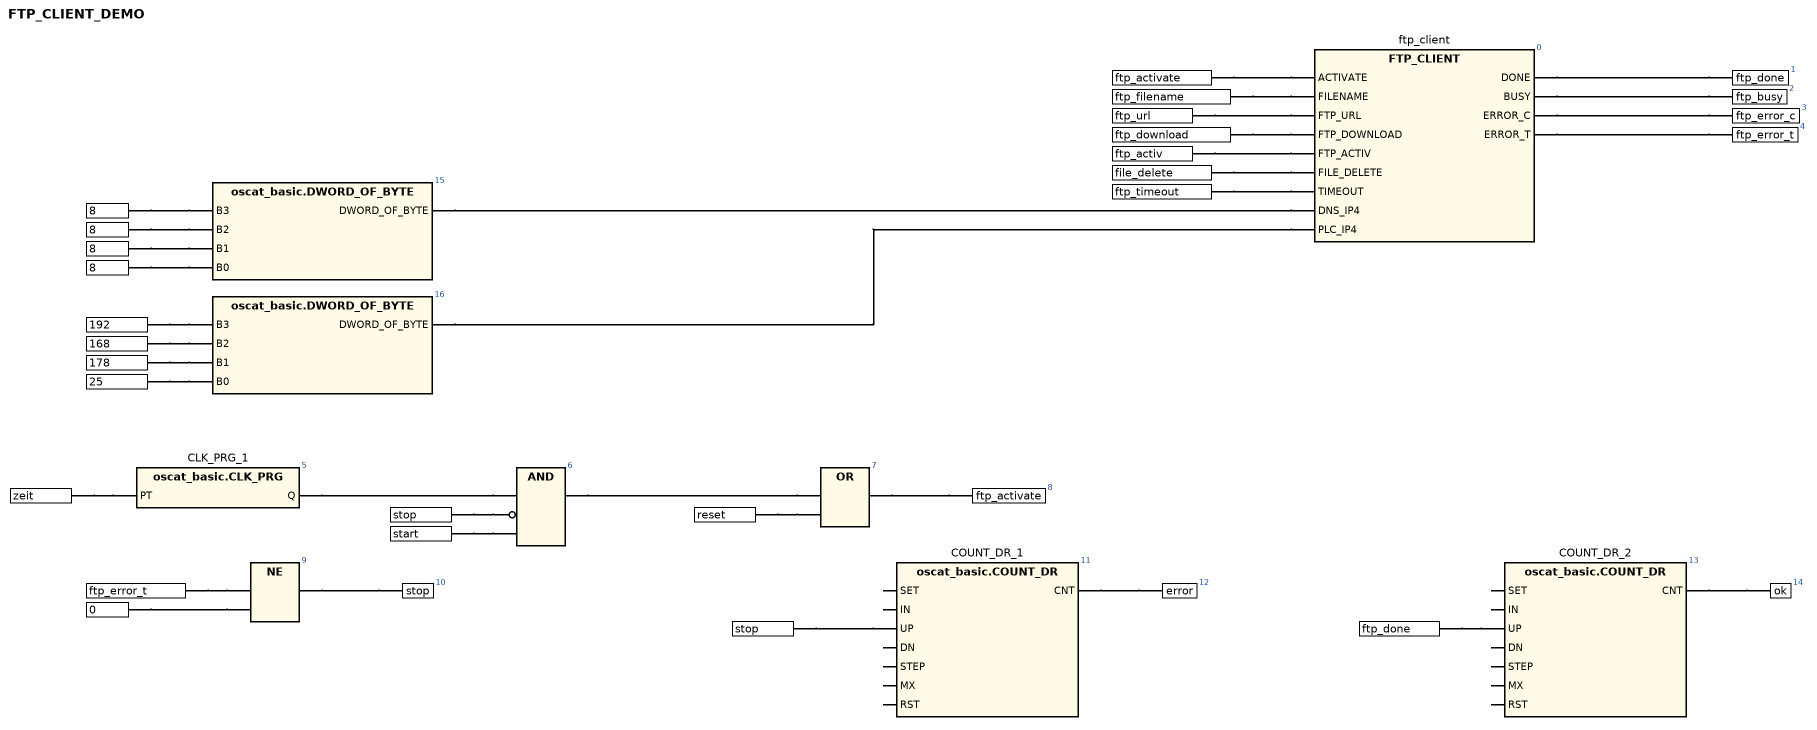
ftp_client(
    ACTIVATE := ftp_activate,
    FILENAME := ftp_filename,
    FTP_URL := ftp_url,
    FTP_DOWNLOAD := ftp_download,
    FTP_ACTIV := ftp_activ,
    FILE_DELETE := file_delete,
    TIMEOUT := ftp_timeout,
    DNS_IP4 := _w1,
    PLC_IP4 := _w2);
ftp_done := ftp_client.DONE;
ftp_busy := ftp_client.BUSY;
ftp_error_c := ftp_client.ERROR_C;
ftp_error_t := ftp_client.ERROR_T;
CLK_PRG_1(PT := zeit); // oscat_basic.CLK_PRG
ftp_activate := CLK_PRG_1.Q AND NOT stop AND start OR reset;
stop := ftp_error_t <> 0;
COUNT_DR_1(UP := stop); // oscat_basic.COUNT_DR
error := COUNT_DR_1.CNT;
COUNT_DR_2(UP := ftp_done); // oscat_basic.COUNT_DR
ok := COUNT_DR_2.CNT;
_w1 := oscat_basic.DWORD_OF_BYTE(B3 := 8, B2 := 8, B1 := 8, B0 := 8);
_w2 := oscat_basic.DWORD_OF_BYTE(B3 := 192, B2 := 168, B1 := 178, B0 := 25);

END_PROGRAM

// POUs/DEMO/GET_WAN_IP_DEMO
PROGRAM GET_WAN_IP_DEMO
VAR
	GET_WAN_IP: GET_WAN_IP;
	IP_C: IP_C;
	S_BUF: NETWORK_BUFFER;
	R_BUF: NETWORK_BUFFER;
	IP_CONTROL_1: IP_CONTROL;
	activate: BOOL;
	done: BOOL;
	error_c: DWORD;
	error_t: BYTE;
	wan_ip: STRING;
	new_ip: BOOL;
END_VAR
VAR // added by the converter: edge detectors and wires of the graphical bodies
    _w1 : ANY;
END_VAR

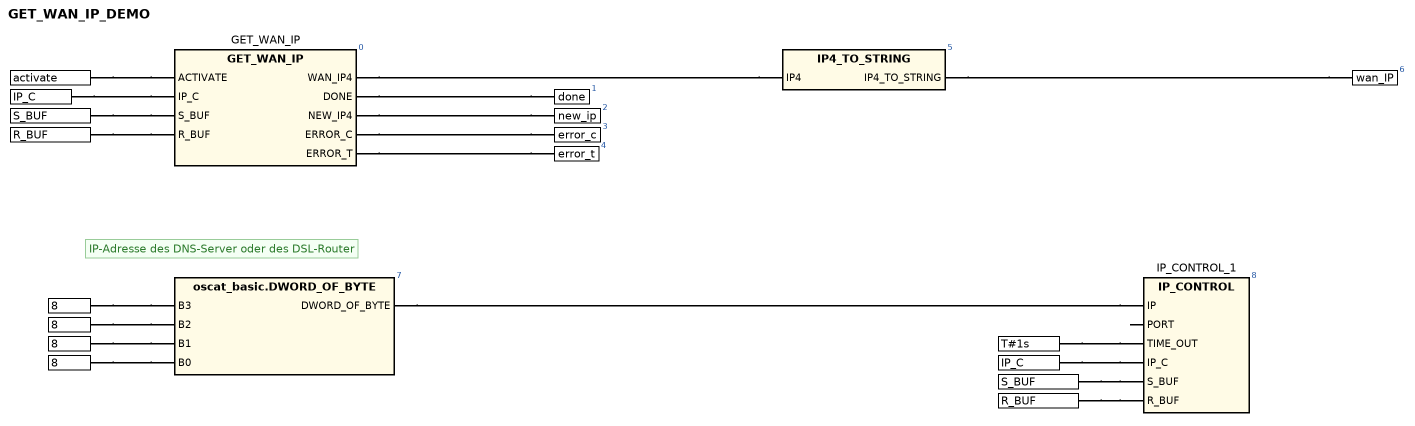
GET_WAN_IP(ACTIVATE := activate, IP_C := IP_C, S_BUF := S_BUF, R_BUF := R_BUF);
done := GET_WAN_IP.DONE;
new_ip := GET_WAN_IP.NEW_IP4;
error_c := GET_WAN_IP.ERROR_C;
error_t := GET_WAN_IP.ERROR_T;
wan_IP := IP4_TO_STRING(IP4 := GET_WAN_IP.WAN_IP4);
// IP-Adresse des DNS-Server oder des DSL-Router
_w1 := oscat_basic.DWORD_OF_BYTE(B3 := 8, B2 := 8, B1 := 8, B0 := 8);
IP_CONTROL_1(IP := _w1, TIME_OUT := T#1s, IP_C := IP_C, S_BUF := S_BUF, R_BUF := R_BUF); // IP_CONTROL

END_PROGRAM

// POUs/CONVERT/HTML_DECODE
FUNCTION HTML_DECODE : STRING(OSCAT_BASIC.STRING_LENGTH)
VAR_INPUT
	IN : STRING(OSCAT_BASIC.STRING_LENGTH);
END_VAR
VAR
	pos : INT;
	end : INT;
	tmp : STRING(10);
	code : STRING(1);
END_VAR

(*
version 1.3		10. may 2010
programmer 	hugo
tested by		oscat

HTML_DECODE converts HTML coded characters to text. 
&amp; is replaced by & ("Ampersand")
&lt; is replaced by < ("lower than")
&gt; is replaced by > ("greater than")
&quot; is replaced by " ("Quote")
all other &names characters are replaced by their respective character codes.

*)

HTML_DECODE := IN;

(* docode characters encoded by character position *)
pos := FIND(HTML_DECODE, '&');
WHILE pos > 0 DO
	tmp := MID(HTML_DECODE, 2, pos + 1);
	IF tmp = '#x' OR tmp = '#X' THEN
		(* hexadecimal representation found *)
		tmp := MID(HTML_DECODE, 10, pos + 3);
		end := FIND(tmp, ';');
		CODE := OSCAT_BASIC.CHR_TO_STRING(DWORD_TO_BYTE(OSCAT_BASIC.HEX_TO_DWORD(LEFT(tmp, end - 1))));
		HTML_DECODE := REPLACE(HTML_DECODE, CODE, end + 3, pos);
	ELSIF LEFT(tmp,1) = '#' THEN
		tmp := MID(HTML_DECODE, 10, pos + 2);
		end := FIND(tmp, ';');
		CODE := OSCAT_BASIC.CHR_TO_STRING(INT_TO_BYTE(STRING_TO_INT(LEFT(tmp, end - 1))));
		HTML_DECODE := REPLACE(HTML_DECODE, CODE, end + 2, pos);
	ELSE
		(* replace all named characters *)
		tmp := MID(HTML_DECODE, 10, pos + 1);
		end := FIND(tmp, ';');
		CODE := OSCAT_BASIC.CHR_TO_STRING(OSCAT_BASIC.CHARCODE(LEFT(tmp, end - 1)));
		HTML_DECODE := REPLACE(HTML_DECODE, CODE, end + 1, pos);
	END_IF;
	(* search for next occurence of encoded characters *)
	pos := OSCAT_BASIC.FINDP(HTML_DECODE, '&', pos + 1);
END_WHILE;



(* revision history
hm	3. mai. 2008	rev 1.0
	original version

hm	16. jun. 2008	rev 1.1
	changed nested call of replace for better compatibility

hm	17. dec. 2008	rev 1.2
	changed function CHR to CHR_TO_STRING

hm	10. may. 2010	rev 1.3
	stringlength 250

*)

END_FUNCTION

// POUs/CONVERT/HTML_ENCODE
FUNCTION HTML_ENCODE : STRING(OSCAT_BASIC.STRING_LENGTH)
VAR_INPUT
	IN : STRING(OSCAT_BASIC.STRING_LENGTH);
	M : BOOL;
END_VAR
VAR
	pt_in : POINTER TO ARRAY[1..255] OF BYTE;
	pt_out : POINTER TO ARRAY[1..256] OF BYTE;
	pos_in : INT;
	pos_out : INT;
	stop : INT;
	B: BYTE;
	tmp : STRING(10);
	i: INT;
END_VAR


(*
version 1.1		10. may. 2010
programmer 	hugo
tested by		hugo 

HTML_ENCODE checks a string if it contains reserved HTML characters and converts them to alternative html coding.
& is replaced by &amp; ("Ampersand")
< is replaced by &lt; ("lower than")
> is replaced by &gt; ("greater than")
" is replaced by &quot; ("Quote")

*)

pt_in  := ADR(in);
pt_out := ADR(HTML_ENCODE);

(* scan the input string and convert unallowed characters *)
pos_in := 1;
stop := LEN(in);
FOR pos_out := 1 TO 250 DO
	IF pos_in > stop THEN EXIT; END_IF;
	B := pt_in^[pos_in];
	CASE BYTE_TO_INT(B) OF
		34: (* " detected *)
			IF pos_out > OSCAT_BASIC.STRING_LENGTH - 6 THEN EXIT; END_IF;
			pt_out^[pos_out] := 38;
			pos_out := pos_out + 1;
			pt_out^[pos_out] := 113;
			pos_out := pos_out + 1;
			pt_out^[pos_out] := 117;
			pos_out := pos_out + 1;
			pt_out^[pos_out] := 111;
			pos_out := pos_out + 1;
			pt_out^[pos_out] := 116;
			pos_out := pos_out + 1;
			pt_out^[pos_out] := 59;
		38: (* & detected *)
			IF pos_out > OSCAT_BASIC.STRING_LENGTH - 5 THEN EXIT; END_IF;
			pt_out^[pos_out] := 38;
			pos_out := pos_out + 1;
			pt_out^[pos_out] := 97;
			pos_out := pos_out + 1;
			pt_out^[pos_out] := 109;
			pos_out := pos_out + 1;
			pt_out^[pos_out] := 112;
			pos_out := pos_out + 1;
			pt_out^[pos_out] := 59;
		60: (* < detected *)
			IF pos_out > OSCAT_BASIC.STRING_LENGTH - 4 THEN EXIT; END_IF;
			pt_out^[pos_out] := 38;
			pos_out := pos_out + 1;
			pt_out^[pos_out] := 108;
			pos_out := pos_out + 1;
			pt_out^[pos_out] := 116;
			pos_out := pos_out + 1;
			pt_out^[pos_out] := 59;
		62: (* > detected *)
			IF pos_out > OSCAT_BASIC.STRING_LENGTH - 4 THEN EXIT; END_IF;
			pt_out^[pos_out] := 38;
			pos_out := pos_out + 1;
			pt_out^[pos_out] := 103;
			pos_out := pos_out + 1;
			pt_out^[pos_out] := 116;
			pos_out := pos_out + 1;
			pt_out^[pos_out] := 59;
	ELSE
		IF M AND B > 127 THEN
			tmp := OSCAT_BASIC.CHARNAME(B);
			(* exit if output string has not enough space *)
			IF pos_out + LEN(tmp) + 2 <= 250 THEN
				pt_out^[pos_out] := 38;
				pos_out := pos_out + 1;
				FOR i := 1 TO LEN(tmp) DO
					pt_out^[pos_out] := OSCAT_BASIC.CODE(tmp, i);
					pos_out := pos_out + 1;
				END_FOR;
				pt_out^[pos_out] := 59;
			END_IF;
		ELSE
			pt_out^[pos_out] := B;
		END_IF;
	END_CASE;
	(* increment in by 1 *)
	pos_in := pos_in + 1;
END_FOR;

(* terminate the output string *)
pt_out^[pos_out] := 0;



(* revision history
hm		3. mai. 2008	rev 1.0
	original version

hm		10. mai. 2008	rev 1.1
	stringlength 250
*)

END_FUNCTION

// POUs/DEMO/HTTP_DEMO
PROGRAM HTTP_DEMO
VAR
	url_text : STRING := 'http://weather.yahooapis.com/forecastrss?p=94089&u=c';
	URL_DATA : URL;
	IP_C: IP_C;
	S_BUF: NETWORK_BUFFER;
	R_BUF: NETWORK_BUFFER;
	IP_CONTROL_1: IP_CONTROL;
	DNS_CLIENT: DNS_CLIENT;
	HTTP_GET: HTTP_GET;
	http_release: BOOL;
	enable: BOOL := TRUE;
	http_status: STRING;
	header_start: UINT;
	header_stop: UINT;
	body_start: UINT;
	body_stop: UINT;
	http_get_done: BOOL;
	http_get_error: DWORD;
	COUNT_DR: OSCAT_BASIC.COUNT_DR;
	cycles: DWORD;
	TON_1: TON;
	F_TRIG: F_TRIG;
END_VAR
VAR // added by the converter: edge detectors and wires of the graphical bodies
    _w1 : ANY;
END_VAR

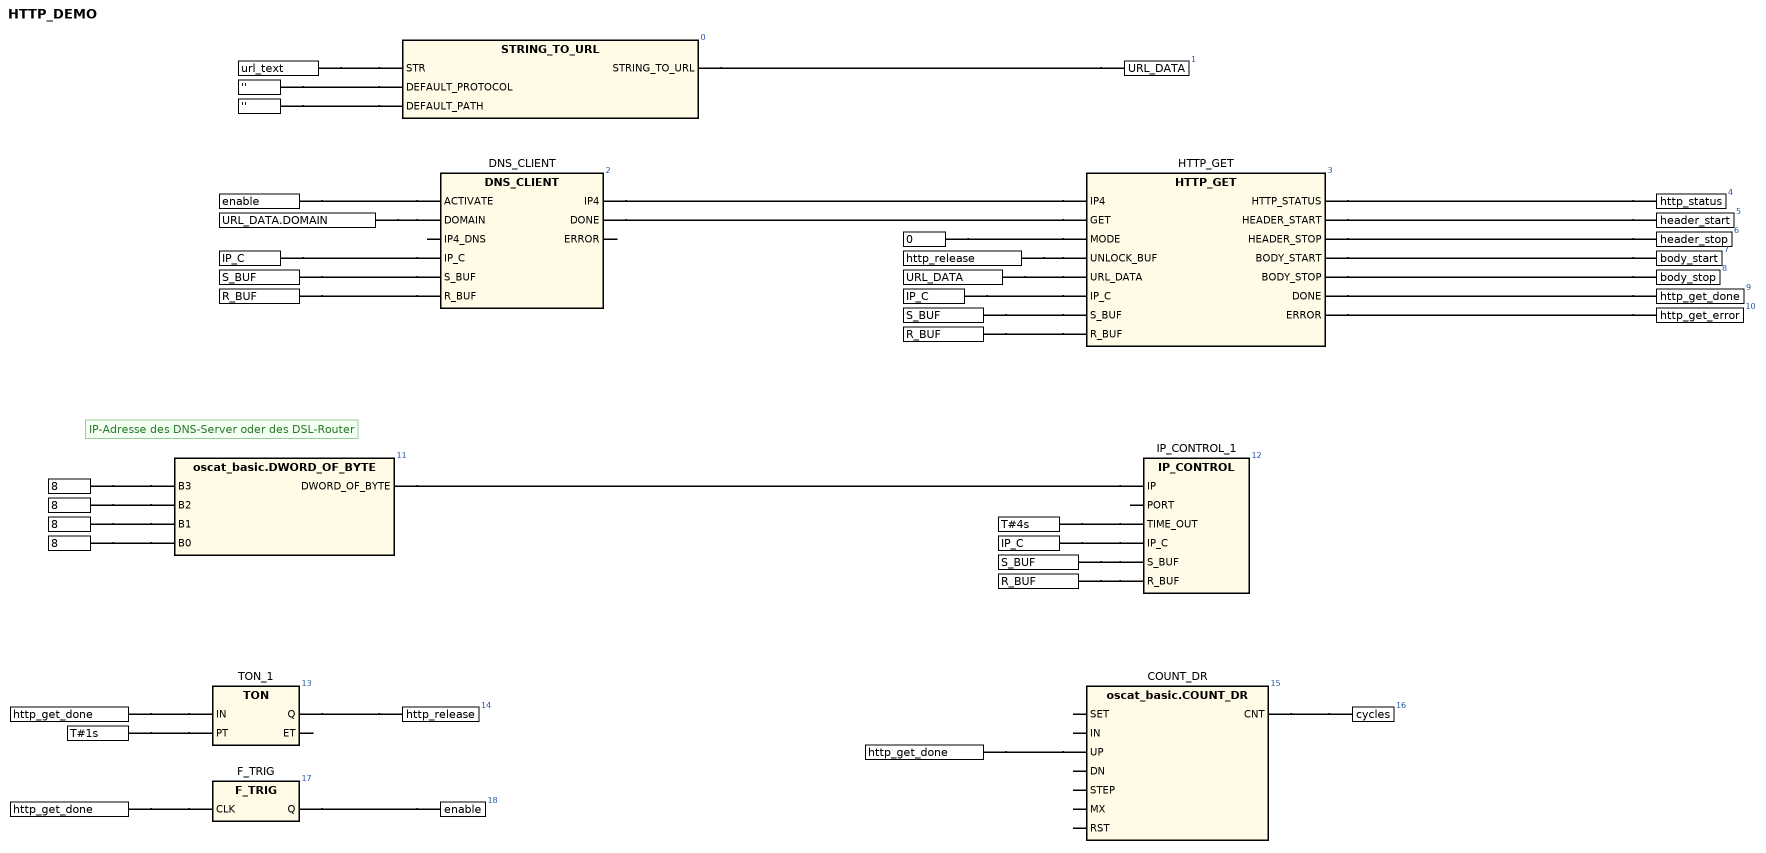
URL_DATA := STRING_TO_URL(STR := url_text, DEFAULT_PROTOCOL := '', DEFAULT_PATH := '');
DNS_CLIENT(ACTIVATE := enable, DOMAIN := URL_DATA.DOMAIN, IP_C := IP_C, S_BUF := S_BUF, R_BUF := R_BUF);
HTTP_GET(
    IP4 := DNS_CLIENT.IP4,
    GET := DNS_CLIENT.DONE,
    MODE := 0,
    UNLOCK_BUF := http_release,
    URL_DATA := URL_DATA,
    IP_C := IP_C,
    S_BUF := S_BUF,
    R_BUF := R_BUF);
http_status := HTTP_GET.HTTP_STATUS;
header_start := HTTP_GET.HEADER_START;
header_stop := HTTP_GET.HEADER_STOP;
body_start := HTTP_GET.BODY_START;
body_stop := HTTP_GET.BODY_STOP;
http_get_done := HTTP_GET.DONE;
http_get_error := HTTP_GET.ERROR;
// IP-Adresse des DNS-Server oder des DSL-Router
_w1 := oscat_basic.DWORD_OF_BYTE(B3 := 8, B2 := 8, B1 := 8, B0 := 8);
IP_CONTROL_1(IP := _w1, TIME_OUT := T#4s, IP_C := IP_C, S_BUF := S_BUF, R_BUF := R_BUF); // IP_CONTROL
TON_1(IN := http_get_done, PT := T#1s); // TON
http_release := TON_1.Q;
COUNT_DR(UP := http_get_done); // oscat_basic.COUNT_DR
cycles := COUNT_DR.CNT;
F_TRIG(CLK := http_get_done);
enable := F_TRIG.Q;

END_PROGRAM

// POUs/FILE/INI_PARSER_BUF
FUNCTION_BLOCK INI_PARSER_BUF
VAR_IN_OUT
	STR : STRING(OSCAT_BASIC.STRING_LENGTH);
	RUN : BYTE;
	OFFSET : UDINT;
	KEY : STRING(OSCAT_BASIC.STRING_LENGTH);
	VALUE : STRING(OSCAT_BASIC.STRING_LENGTH);
	PT : NETWORK_BUFFER;
END_VAR
VAR_OUTPUT
	RESULT : BYTE;
END_VAR
VAR
	step : INT;
	size : INT;
	c : BYTE;
	k_add : BYTE;
	v_add : BYTE;
	i : INT;
	state : BYTE;
	eof : BOOL;
	pv : POINTER TO BYTE;
	pk : POINTER TO BYTE;
	pve : DWORD;
	pke : DWORD;
	watchdog : TON;

	(*LOG_MSG : LOG_MSG;
	_debug_enable : BOOL := TRUE;
	step_last : INT;*)
END_VAR

(*
version 1.0		23. sep. 2010
programmer 		ks
tested by			ks

INI_PARSER_BUF liefert die Elemente einer Initialisierungsdatei die in einem Bytearray abgelegt ist.

--------------------------------------

RUN Mode
00 = kein Befehl aktiv
01 = Section melden
02 = Key melden
03 = Section oder Key melden

Result Codes
01 = Section gefunden
02 = Key gefunden
05 = Befehl in Arbeit (Busy)
10 = nichts gefunden - Daten-Ende erreicht
11 = keinen Key gefunden - Section-Ende erreicht

State Codes
00 = Indexüberschreitung - Bufferende
01 = Section gefunden
02 = Key gefunden
03 = Kommentar gefunden
05 = Befehl in Arbeit (Busy)
10 = nichts gefunden - Daten-Ende erreicht

*)

IF RUN > 0 THEN
	IF state = 0 THEN (* Auswertung neu beginnen *)

		pv := ADR(VALUE);
		pv^ := 0; (* VALUE = '' *)
		pve := pv + INT_TO_DWORD(OSCAT_BASIC.STRING_LENGTH);
		pk := ADR(KEY);
		pk^ := 0; (* KEY = '' *)
		pke := pk + INT_TO_DWORD(OSCAT_BASIC.STRING_LENGTH);

		i := UDINT_TO_INT(OFFSET);
		size := UINT_TO_INT(PT.SIZE) - 1;
		RESULT := 0;
		state := 5; (* Befehl in Arbeit (Busy) *)
		step := 0; (* Auswertung neu beginnen *)

		(*####################  DEBUG-MESSAGE  ###################################*)
		(*IF _debug_enable THEN
			LOG_CL.NEW_MSG := 'IPB: Startindex: ~1';
			LOG_CL.PRINTF[1]  := INT_TO_STRING(i);
			LOG_MSG();
		END_IF;*)
		(*########################################################################*)
	END_IF;

	watchdog(IN:=FALSE,PT:=T#1ms); (* Timer neustarten *)
	watchdog.IN := TRUE;

	WHILE (state = 5) DO (* Schleife solange kein Ergebnis *)

		watchdog(); (* Timer aktualisieren *)

		IF watchdog.Q THEN (* watchdog ausgelöst *)
			state := 5;
			EXIT;
		ELSIF i > size THEN (* kein weiteres zeichen vorhanden *)
			state := 10; (* nichts gefunden - Daten-Ende erreicht *)
			EXIT;
		ELSE

			c := PT.BUFFER[i]; (* neues Zeichen aus Buffer lesen *)
			eof := i + 1 = PT.SIZE; (* End of File *)

			k_add := 0;
			v_add := 0;

			CASE step OF

			0: (* noch kein Modus erkannt *)
				IF c = 91 THEN (* mit "[" vergleichen *)
					step := 200; (* Modus für Section aktivieren *)
				ELSIF c = 59 OR c = 35 THEN (* mit ";" und '#' vergleichen *)
					step := 100; (* Modus für Kommentar aktivieren *)
				ELSIF c > 32 THEN (* Key erkannt *)
					k_add := c; (* Zeichen ablegen *)
					step := 300; (* Key auswertung starten *)
				END_IF;
			100: (* Kommentar erkannt -> Zeilenende suchen *)
				IF c < 32 THEN (* prüfe auf Steuerzeichen *)
					state  := 3; (* Beenden -> Kommentar wurde gefunden *)
				END_IF;
			200: (* Sections-start erkannt -> Sectionsende suchen *)
				IF c = 93 THEN (* mit "]" vergleichen *)
					IF pk > ADR(KEY) > 0 THEN (* innerhalb von [] muss sich mindestens ein Zeichen befinden *)
						state  := 1; (* Beenden -> Section wurde gefunden *)
					ELSE
						pk := ADR(KEY);
						pk^ := 0; (* KEY = '' *)
						step := 0; (* fehlerhafte Section-Zeile vorhanden -> weitersuchen *)
					END_IF;
				ELSIF c < 32 OR eof THEN (* Steuerzeichen - fehlerhafte Section-Zeile -> weitersuchen *)
					pk := ADR(KEY);
					pk^ := 0; (* KEY = '' *)
					step := 0;
				ELSE
					k_add := c; (* Zeichen ablegen *)
				END_IF;
			300: (* Beginn: Key erkannt -> Name auswerten *)
				IF c < 32 THEN (* Steuerzeichen - fehlerhafte Key-Zeile -> weitersuchen *)
					pk := ADR(KEY);
					pk^ := 0; (* KEY = '' *)
					step := 0;
				ELSIF c = 61 THEN (* prüfe auf '=' *)
					step := 330;
				ELSE
					k_add := c; (* Zeichen ablegen *)
				END_IF;
			330: (* KeyValue beginn suchen *)
				IF c < 32 THEN (* Steuerzeichen  *)
					state := 2; (* Key ohne Value gefunden *)
				ELSIF eof THEN
					state := 2; (* Key ohne Value gefunden *)
					v_add := c; (* Zeichen ablegen *)
				ELSE
					v_add := c; (* Zeichen ablegen *)
					step := 350;
				END_IF;
			350: (* KeyValue Ende suchen *)
				IF c < 32 THEN (* Steuerzeichen *)
					state := 2; (* Key gefunden *)
				ELSIF eof THEN
					v_add := c; (* Zeichen ablegen *)
					state := 2; (* Key gefunden *)
				ELSE
					v_add := c; (* Zeichen ablegen *)
				END_IF;
			END_CASE;

			IF v_add > 0  AND pv < pve THEN (* Zeichen zu Value-String hinzufügen *)
				pv^ := v_add; (* Zeichen eintragen *)
				pv := pv + 1;
				pv^ := 0; (* String-Terminierung eintragen *)
			END_IF;

			IF k_add > 0 AND pk < pke THEN (* Zeichen zu Key-String hinzufügen *)
				pk^ := k_add; (* Zeichen eintragen *)
				pk := pk + 1;
				pk^ := 0; (* String-Terminierung eintragen *)
			END_IF;

			i := i + 1; (* Datenzeiger erhöhen *)

		END_IF;
	END_WHILE;

	CASE state OF
	01:	(* Section gefunden *)
		IF RUN = 1 OR RUN = 3 THEN (* Section vorgewählt oder alles rückmelden *)
			IF KEY = STR OR LEN(STR) = 0 THEN (* mit gesuchter Section vergleichen oder keine Section vorgegeben *)
				RESULT := 1; (* Section gefunden *)
				OFFSET := i; (* Offset uebernehmen *)
				RUN := 0;
				state := 0;
			END_IF;
		ELSE
			pk := ADR(KEY);
			pk^ := 0; (* KEY = '' *)
			RESULT := 11; (* Key nicht gefunden , Section-Ende - Offset nicht verändern *)
			RUN := 0;
			state := 0;
		END_IF;
	02:	(* Key gefunden *)
		IF RUN = 2 OR RUN = 3 THEN (* Key vorgewählt oder alles rückmelden *)
			IF KEY = STR OR LEN(STR) = 0 THEN (* mit gesuchten Key vergleichen *)
				RESULT := 2; (* Key gefunden *)
				OFFSET := i; (* Offset uebernehmen *)
				RUN := 0;
				state := 0;
			END_IF;
		END_IF;
	03:	(* Kommenar gefunden *)
		OFFSET := i; (* Offset uebernehmen *)
		state := 0;

	05:	RESULT := 5; (* in Arbeit *)

	10:	(* Indexüberschreitung - Bufferende *)
		RESULT := 10; (* nichts gefunden - Datenende erreicht *)
		OFFSET := i; (* Offset uebernehmen *)
		RUN := 0;
		state := 0;
	END_CASE;

	(*####################  DEBUG-MESSAGE  ###################################*)
	(*IF _debug_enable THEN
		LOG_CL.NEW_MSG := 'IPF: intern Result ~1 , state ~2, step ~3 , offset ~4, run ~5';
		LOG_CL.PRINTF[1] := BYTE_TO_STRING(RESULT);
		LOG_CL.PRINTF[2] := BYTE_TO_STRING(state);
		LOG_CL.PRINTF[3] := INT_TO_STRING(step);
		LOG_CL.PRINTF[4] := UDINT_TO_STRING(OFFSET);
		LOG_CL.PRINTF[5] := BYTE_TO_STRING(RUN);
		LOG_MSG();
	END_IF;*)
	(*########################################################################*)

END_IF;

(*####################  DEBUG-MESSAGE  ###################################*)
(*IF _debug_enable THEN
	IF step_last <> step THEN
		LOG_CL.NEW_MSG := 'IPB: Step: ~1';
		LOG_CL.PRINTF[1]  := INT_TO_STRING(step);
		LOG_MSG();
	END_IF;
	step_last := step;
END_IF;*)
(*########################################################################*)

(* revision history
ks	23. sep. 2010	rev 1.0
	original version
*)

END_FUNCTION_BLOCK

// POUs/DEMO/INI_PARSER_BUF_DEMO
PROGRAM INI_PARSER_BUF_DEMO
VAR
	STATION_NAME : STRING;
	STATION_IP : STRING;
	SMTP_SERVER : STRING;
	SMTP_FROM :	STRING;

	IPB : INI_PARSER_BUF;
	FS : FILE_SERVER;
	FSD : FILE_SERVER_DATA;
	PT : NETWORK_BUFFER;
	section : INT;
	key : STRING(OSCAT_BASIC.STRING_LENGTH);
	value : STRING(OSCAT_BASIC.STRING_LENGTH);
	str : STRING(OSCAT_BASIC.STRING_LENGTH);
	step : INT;
	result : BYTE;
	offset : UDINT;
	run : BYTE;
	done : BOOL;

	(*_debug_enable : BOOL := TRUE;
	LOG_MSG : LOG_MSG;*)
END_VAR

(* Demo-Programm: INI-Datei mittels Enumeration auswerten *)

(* ----- den nachfolgenden Textblock als datei "config.ini" auf der sps ablegen ---
# Demo - Initialisierungsdatei

[Station]
NAME=Test_Station_1
IP=192.168.178.1

[SMTP]
SERVER=test.server.de
FROM=test1@gmx.net
---------------------------------------------------------------------------------*)

CASE step OF

00:	IF NOT done THEN
	 	(* File_Daten einrichten  *)
		FSD.FILENAME := 'config.ini'; (* Dateiname *)
		FSD.MODE := 1; (* vorhandene Datei zum lesen öffnen *)
		FSD.OFFSET := 0; (* Start bei Dateianfang *)
		PT.SIZE := 65535; (* maximale länge einlesen *)
		step := 10;
	END_IF;

10:	IF FSD.MODE = 0 THEN (* Datei geöffnet ? *)
		OFFSET := 0; (* Start Offset vorgeben *)
		str := '';
		run := 3; (* key suchen *)
		step := 20;
	END_IF;

20:	IF run = 0 THEN
		(* ---------------------- Debug-Message ----------------------------*)
		(*IF _debug_enable THEN
			LOG_CL.NEW_MSG := 'IPBD: /key >~1< /value >~2< /offset ~3 /Run ~4 /Result ~5';
			LOG_CL.PRINTF[1] := key;
			LOG_CL.PRINTF[2] := value;
			LOG_CL.PRINTF[3] := UDINT_TO_STRING(OFFSET);
			LOG_CL.PRINTF[4] := BYTE_TO_STRING(run);
			LOG_CL.PRINTF[5] := BYTE_TO_STRING(result);
			LOG_MSG();
		END_IF;*)
		(* -----------------------------------------------------------------*)

		run := 3; (* vorbelegung -> naechsten key suchen *)

		IF result = 1 THEN (* neue Sektion gefunden *)
			IF key = 'Station' THEN
				section := 1;
			ELSIF key = 'SMTP' THEN
				section := 2;

			(* hier können weitere Section hinzugefügt werden *)

			ELSE
				section := 0; (* unbekannte sektion gefunden -> ignorieren *)
			END_IF;

		ELSIF result = 2 AND section > 0 THEN (* Key in einer bekannten sektion gefunden *)

			CASE section OF

			1:  (* Section: Station *)
				IF key = 'NAME' THEN
					STATION_NAME := value; (* Name *)
				ELSIF key = 'IP' THEN
					STATION_IP := value; (* IP-Adresse *)
				END_IF;

				(* hier können weitere Schlüsselsauswertungen hinzugefügt werden *)

			2:  (* Section: SMTP *)
				IF key = 'SERVER' THEN
					SMTP_SERVER := value; (* SMTP Server *)
				ELSIF key = 'FROM' THEN
					SMTP_FROM := value; (* SMTP Absender *)
				END_IF;

				(* hier können weitere Schlüsselsauswertungen hinzugefügt werden *)

			END_CASE;

		ELSIF result = 10 THEN (* nichts mehr gefunden *)
			run := 0; (* keine weitere INI Auswertung erwünscht *)
			FSD.MODE := 5; (* Datei schliessen *)
			step := 30;
		END_IF;
	END_IF;

30:	IF FSD.MODE = 0 THEN (* Datei geschlossen ? *)
		step := 0;
		done := TRUE;
	END_IF;

END_CASE;

IPB(STR:=str,RUN:=run,OFFSET:=OFFSET,KEY:=key,VALUE:=value,PT:=PT); (* INI PARAMETER BUF *)
result:=IPB.RESULT;

FS(FSD:=FSD,PT:=PT); (* FILE_SERVER *)

END_PROGRAM

// POUs/FILE/INI_PARSER_FILE
FUNCTION_BLOCK INI_PARSER_FILE
VAR_IN_OUT
	FILENAME : STRING;
	FSD : FILE_SERVER_DATA	;
	STR : STRING(OSCAT_BASIC.STRING_LENGTH);
	RUN : BYTE;
	OFFSET : UDINT;
	KEY : STRING(OSCAT_BASIC.STRING_LENGTH);
	VALUE : STRING(OSCAT_BASIC.STRING_LENGTH);
	PT	: NETWORK_BUFFER;
END_VAR
VAR_OUTPUT
	RESULT : BYTE;
END_VAR
VAR
	FB : FILE_BLOCK;
	i : UDINT;
	state : BYTE;
	e : BYTE;
	mode : BYTE;
	step : INT;
	c : BYTE;
	k_add : BYTE;
	v_add : BYTE;
	eof : BOOL;
	pv : POINTER TO BYTE;
	pk : POINTER TO BYTE;
	pve : DWORD;
	pke : DWORD;
	watchdog : TON;

	(*LOG_MSG : LOG_MSG;
	_debug_enable : BOOL := TRUE;
	step_last : INT;*)
END_VAR

(*
version 1.0		23. sep. 2010
programmer 		ks
tested by			ks

INI_PARSER_FILE liefert die Elemente einer Initialisierungsdatei.

--------------------------------------

RUN Mode
00 = kein Befehl aktiv
01 = Section melden
02 = Key melden
03 = Section oder Key melden

Result Codes
01 = Section gefunden
02 = Key gefunden
05 = Befehl in Arbeit (Busy)
10 = nichts gefunden - Daten-Ende erreicht
11 = keinen Key gefunden - Section-Ende erreicht

State Codes
00 = Indexüberschreitung - Bufferende
01 = Section gefunden
02 = Key gefunden
03 = Kommentar gefunden
05 = Befehl in Arbeit (Busy)
10 = nichts gefunden - Daten-Ende erreicht

*)

IF RUN > 0 THEN

	IF state = 0 THEN (* Auswertung neu beginnen *)
		pv := ADR(VALUE);
		pv^ := 0; (* VALUE = '' *)
		pve := pv + INT_TO_DWORD(OSCAT_BASIC.STRING_LENGTH);
		pk := ADR(KEY);
		pk^ := 0; (* KEY = '' *)
		pke := pk + INT_TO_DWORD(OSCAT_BASIC.STRING_LENGTH);

		i := OFFSET;
		RESULT := 0;
		state := 5; (* Befehl in Arbeit (Busy) *)
		step := 0; (* Auswertung neu beginnen *)

		(*####################  DEBUG-MESSAGE  ###################################*)
		(*IF _debug_enable THEN
			LOG_CL.NEW_MSG := 'IPF: Startindex: ~1';
			LOG_CL.PRINTF[1] := UDINT_TO_STRING(i);
			LOG_MSG();
		END_IF;*)
		(*########################################################################*)

	END_IF;

	watchdog(IN:=FALSE,PT:=T#1ms); (* Timer neustarten *)
	watchdog.IN := TRUE;

	WHILE (state = 5) DO (* Schleife solange kein Ergebnis *)

		mode := 1;
		FB(MODE:=mode,FSD:=fsd,PT:=PT,FILENAME:=FILENAME,POS:=i );
		e:=FB.ERROR;
		c:=FB.DATA;

		eof := i + 1 = FSD.FILE_SIZE; (* End of File *)

		(*####################  DEBUG-MESSAGE  ###################################*)
		(*IF _debug_enable THEN
			LOG_CL.NEW_MSG := 'IPF: mode: ~1, error: ~2 , >~7<>~3< ~4 step ~5 index ~6';
			LOG_CL.PRINTF[1] := BYTE_TO_STRING(mode);
			LOG_CL.PRINTF[2] := BYTE_TO_STRING(e);
			LOG_CL.PRINTF[3] := BYTE_TO_STRING(c);
			LOG_CL.PRINTF[4] := BOOL_TO_STRING(eof);
			LOG_CL.PRINTF[5] := INT_TO_STRING(step);
			LOG_CL.PRINTF[6] := UDINT_TO_STRING(i);
			LOG_CL.PRINTF[7] := CHR_TO_STRING(c);
			LOG_MSG();
		END_IF;*)
		(*########################################################################*)

		watchdog(); (* Timer aktualisieren *)

		IF mode > 0 OR watchdog.Q THEN (* Baustein noch aktiv, oder watchdog ausgelöst *)
			state := 5;
			EXIT;
		ELSIF e > 0 THEN (* File_error oder kein weiteres zeichen vorhanden *)
			state := 10; (* nichts gefunden - Daten-Ende erreicht *)
			EXIT;
		ELSE

			k_add := 0;
			v_add := 0;

			CASE step OF

			0: (* noch kein Modus erkannt *)
				IF c = 91 THEN (* mit "[" vergleichen *)
					step := 200; (* Modus für Section aktivieren *)
				ELSIF c = 59 OR c = 35 THEN (* mit ";" und '#' vergleichen *)
					step := 100; (* Modus für Kommentar aktivieren *)
				ELSIF c > 32 THEN (* Key erkannt *)
					k_add := c; (* Zeichen ablegen *)
					step := 300; (* Key auswertung starten *)
				END_IF;
			100: (* Kommentar erkannt -> Zeilenende suchen *)
				IF c < 32 THEN (* prüfe auf Steuerzeichen *)
					state  := 3; (* Beenden -> Kommentar wurde gefunden *)
				END_IF;
			200: (* Sections-start erkannt -> Sectionsende suchen *)
				IF c = 93 THEN (* mit "]" vergleichen *)
					IF pk > ADR(KEY) > 0 THEN (* innerhalb von [] muss sich mindestens ein Zeichen befinden *)
						state  := 1; (* Beenden -> Section wurde gefunden *)
					ELSE
						pk := ADR(KEY);
						pk^ := 0; (* KEY = '' *)
						step := 0; (* fehlerhafte Section-Zeile vorhanden -> weitersuchen *)
					END_IF;
				ELSIF c < 32 OR eof THEN (* Steuerzeichen - fehlerhafte Section-Zeile -> weitersuchen *)
					pk := ADR(KEY);
					pk^ := 0; (* KEY = '' *)
					step := 0;
				ELSE
					k_add := c; (* Zeichen ablegen *)
				END_IF;
			300: (* Beginn: Key erkannt -> Name auswerten *)
				IF c < 32 THEN (* Steuerzeichen - fehlerhafte Key-Zeile -> weitersuchen *)
					pk := ADR(KEY);
					pk^ := 0; (* KEY = '' *)
					step := 0;
				ELSIF c = 61 THEN (* prüfe auf '=' *)
					step := 330;
				ELSE
					k_add := c; (* Zeichen ablegen *)
				END_IF;
			330: (* KeyValue beginn suchen *)
				IF c < 32 THEN (* Steuerzeichen  *)
					state := 2; (* Key ohne Value gefunden *)
				ELSIF eof THEN
					state := 2; (* Key ohne Value gefunden *)
					v_add := c; (* Zeichen ablegen *)
				ELSE
					v_add := c; (* Zeichen ablegen *)
					step := 350;
				END_IF;
			350: (* KeyValue Ende suchen *)
				IF c < 32 THEN (* Steuerzeichen *)
					state := 2; (* Key gefunden *)
				ELSIF eof THEN
					v_add := c; (* Zeichen ablegen *)
					state := 2; (* Key gefunden *)
				ELSE
					v_add := c; (* Zeichen ablegen *)
				END_IF;
			END_CASE;

			IF v_add > 0  AND pv < pve THEN (* Zeichen zu Value-String hinzufügen *)
				pv^ := v_add; (* Zeichen eintragen *)
				pv := pv + 1;
				pv^ := 0; (* String-Terminierung eintragen *)
			END_IF;

			IF k_add > 0 AND pk < pke THEN (* Zeichen zu Key-String hinzufügen *)
				pk^ := k_add; (* Zeichen eintragen *)
				pk := pk + 1;
				pk^ := 0; (* String-Terminierung eintragen *)
			END_IF;

			i := i + 1; (* Datenzeiger erhöhen *)

		END_IF;
	END_WHILE;

	CASE state OF
	01:	(* Section gefunden *)
		IF RUN = 1 OR RUN = 3 THEN (* Section vorgewählt oder alles rückmelden *)
			IF KEY = STR OR LEN(STR) = 0 THEN (* mit gesuchter Section vergleichen oder keine Section vorgegeben *)
				RESULT := 1; (* Section gefunden *)
				OFFSET := i; (* Offset uebernehmen *)
				RUN := 0;
				state := 0;
			END_IF;
		ELSE
			pk := ADR(KEY);
			pk^ := 0; (* KEY = '' *)
			RESULT := 11; (* Key nicht gefunden , Section-Ende - Offset nicht verändern *)
			RUN := 0;
			state := 0;
		END_IF;
	02:	(* Key gefunden *)
		IF RUN = 2 OR RUN = 3 THEN (* Key vorgewählt oder alles rückmelden *)
			IF KEY = STR OR LEN(STR) = 0 THEN (* mit gesuchten Key vergleichen *)
				RESULT := 2; (* Key gefunden *)
				OFFSET := i; (* Offset uebernehmen *)
				RUN := 0;
				state := 0;
			END_IF;
		END_IF;
	03:	(* Kommenar gefunden *)
		OFFSET := i; (* Offset uebernehmen *)
		state := 0;

	05:	RESULT := 5; (* in Arbeit *)

	10:	(* Indexüberschreitung - Bufferende *)
		RESULT := 10; (* nichts gefunden - Datenende erreicht *)
		OFFSET := i; (* Offset uebernehmen *)
		RUN := 0;
		state := 0;
	END_CASE;

	(*####################  DEBUG-MESSAGE  ###################################*)
	(*IF _debug_enable THEN
		LOG_CL.NEW_MSG := 'IPF: intern Result ~1 , state ~2, step ~3 , offset ~4, run ~5';
		LOG_CL.PRINTF[1] := BYTE_TO_STRING(RESULT);
		LOG_CL.PRINTF[2] := BYTE_TO_STRING(state);
		LOG_CL.PRINTF[3] := INT_TO_STRING(step);
		LOG_CL.PRINTF[4] := UDINT_TO_STRING(OFFSET);
		LOG_CL.PRINTF[5] := BYTE_TO_STRING(RUN);
		LOG_MSG();
	END_IF;*)
	(*########################################################################*)

END_IF;

(*####################  DEBUG-MESSAGE  ###################################*)
(*IF _debug_enable THEN
	IF step_last <> step THEN
		LOG_CL.NEW_MSG := 'IPB: Step: ~1';
		LOG_CL.PRINTF[1]  := INT_TO_STRING(step);
		LOG_MSG();
	END_IF;
	step_last := step;
END_IF;*)
(*########################################################################*)

(* revision history
ks	23. sep. 2010	rev 1.0
	original version
*)

END_FUNCTION_BLOCK

// POUs/DEMO/INI_PARSER_FILE_DEMO
PROGRAM INI_PARSER_FILE_DEMO
VAR
	STATION_NAME : STRING;
	STATION_IP : STRING;
	SMTP_SERVER : STRING;
	SMTP_FROM : STRING;

	IPF : INI_PARSER_FILE;
	FS : FILE_SERVER;
	FSD : FILE_SERVER_DATA;
	PT : NETWORK_BUFFER;
	section : INT;
	filename : STRING;
	key : STRING(OSCAT_BASIC.STRING_LENGTH);
	value :	STRING(OSCAT_BASIC.STRING_LENGTH);
	str : STRING(OSCAT_BASIC.STRING_LENGTH);
	step : INT;
	result : BYTE;
	offset : UDINT;
	run : BYTE;
	done : BOOL;

	(*LOG_MSG : LOG_MSG;
	_debug_enable : BOOL := TRUE;*)
END_VAR

(* Demo-Programm: INI-Datei mittels Enumeration auswerten *)

(* ----- den nachfolgenden Textblock als datei "config.ini" auf der sps ablegen ---
# Demo - Initialisierungsdatei

[Station]
NAME=Test_Station_1
IP=192.168.178.1

[SMTP]
SERVER=test.server.de
FROM=test1@gmx.net
---------------------------------------------------------------------------------*)

CASE step OF

00:	IF NOT done THEN
		filename := 'config.ini'; (* File_Daten einrichten *)
		OFFSET := 0; (* Start Offset vorgeben *)
		str := '';
		run := 3; (* key suchen *)
		step := 20;
	END_IF;

20:	IF run = 0 THEN (* kein Befehl mehr aktiv ? *)
		(* ---------------------- Debug-Message ----------------------------*)
		(*IF _debug_enable THEN
			LOG_CL.NEW_MSG := 'IPFD: /key >~1< /value >~2< /offset ~3 /Run ~4 /Result ~5';
			LOG_CL.PRINTF[1] := key;
			LOG_CL.PRINTF[2] := value;
			LOG_CL.PRINTF[3] := UDINT_TO_STRING(OFFSET);
			LOG_CL.PRINTF[4] := BYTE_TO_STRING(run);
			LOG_CL.PRINTF[5] := BYTE_TO_STRING(result);
			LOG_MSG();
		END_IF;*)
		(* -----------------------------------------------------------------*)

		run := 3; (* vorbelegung -> naechsten key suchen *)

		IF result = 1 THEN (* neue Sektion gefunden *)
			IF key = 'Station' THEN
				section := 1;
			ELSIF key = 'SMTP' THEN
				section := 2;

			(* hier können weitere Section hinzugefügt werden *)

			ELSE
				section := 0; (* unbekannte sektion gefunden -> ignorieren *)
			END_IF;

		ELSIF result = 2 AND section > 0 THEN (* Key in einer bekannten sektion gefunden *)

			CASE section OF

			1:  (* Section: Station *)
				IF key = 'NAME' THEN
					STATION_NAME := value; (* Name *)
				ELSIF key = 'IP' THEN
					STATION_IP := value; (* IP-Adresse *)
				END_IF;

				(* hier können weitere Schlüsselsauswertungen hinzugefügt werden *)

			2:  (* Section: SMTP *)
				IF key = 'SERVER' THEN
					SMTP_SERVER := value; (* SMTP Server *)
				ELSIF key = 'FROM' THEN
					SMTP_FROM := value; (* SMTP Absender *)
				END_IF;

				(* hier können weitere Schlüsselsauswertungen hinzugefügt werden *)

			END_CASE;

		ELSIF result = 10 THEN (* nichts mehr gefunden *)
			run := 0; (* keine weitere INI Auswertung erwünscht *)
			FSD.MODE := 5; (* Datei schliessen *)
			step := 30;
		END_IF;
	END_IF;

30:	IF FSD.MODE = 0 THEN (* Befehl Datei schliessen beendet *)
		step := 0;
		done := TRUE;
	END_IF;

END_CASE;

IPF(FILENAME:=FILENAME,FSD:=FSD,STR:=str,RUN:=run,OFFSET:=OFFSET,KEY:=key,VALUE:=value,PT:=PT); (* INI PARAMETER FILE *)
result:=IPF.RESULT;

FS(FSD:=FSD,PT:=PT); (* FILE_SERVER *)

END_PROGRAM

// POUs/NETWORK/IP2GEO
FUNCTION_BLOCK IP2GEO
VAR_IN_OUT
	IP_C : IP_C; (* IP_Control Verwaltungsstruktur *)
	S_BUF : NETWORK_BUFFER;
	R_BUF : NETWORK_BUFFER;
	GEO : IP2GEO_DATA;
END_VAR
VAR_INPUT
	IP : DWORD;
	ACTIVATE : BOOL;
END_VAR
VAR_OUTPUT
	BUSY : BOOL;
	DONE : BOOL;
	ERROR_C : DWORD;
	ERROR_T : BYTE;
END_VAR
VAR
	CTRL : XML_CONTROL;
	XML_READER : XML_READER;
	URL_DATA : url;
	DNS_CLIENT : DNS_CLIENT;
	HTTP_GET : HTTP_GET;
	last_state : BOOL;
	value_int :	INT;
	value_real : REAL;
	v_real : REAL;
	state : INT;
END_VAR
(*

version 	1.1	07.oct. 2010
programmer 	ks
tested by	ks

IP2GEO ermittelt die aktuelle WAN-IP und die dazugehörigen geographischen Infos

zusatzinfos: http://www.worldtimezone.com/time/wtzresult.php?CiID=10182&forma=

example:

http://ipinfodb.com/ip_query.php?timezone=true&IP=

<?xml version="1.0" encoding="UTF-8" ?> 
- <Response>
  <Ip>85.127.218.109</Ip> 
  <Status>OK</Status> 
  <CountryCode>AT</CountryCode> 
  <CountryName>Austria</CountryName> 
  <RegionCode>09</RegionCode> 
  <RegionName>Wien</RegionName> 
  <City>Vienna</City> 
  <ZipPostalCode /> 
  <Latitude>48.2</Latitude> 
  <Longitude>16.3667</Longitude> 
  <TimezoneName>Europe/Vienna</TimezoneName> 
  <Gmtoffset>7200</Gmtoffset> 
  <Isdst>1</Isdst> 
  </Response>

*)

CASE state OF

00:
	IF ACTIVATE AND NOT last_state THEN
		state := 20;
		DONE := FALSE;
		BUSY := TRUE;
		ERROR_C := DWORD#0;
		ERROR_T := BYTE#0;
	END_IF;

20: (* URL for DNS UND HTTP-GET *)
	(* Example: http://ipinfodb.com/ip_query.php?ip=10.10.10.10 *)
	(* Example: http://ipinfodb.com/ip_query.php?timezone=true&IP=*)
	URL_DATA:=STRING_TO_URL(STR:='http://ipinfodb.com/ip_query.php?timezone=true&IP=',DEFAULT_PROTOCOL:='',DEFAULT_PATH:='');

	IF IP > DWORD#0 THEN
		URL_DATA.QUERY := CONCAT(URL_DATA.QUERY,IP4_TO_STRING(IP4:=IP));
	END_IF;

	state := 40;

40:
	IF DNS_CLIENT.DONE THEN
		state := 60;
	ELSIF (DNS_CLIENT.ERROR > DWORD#00) THEN
		(* Fehlerbehandlung *)
		ERROR_C := DNS_CLIENT.ERROR;
		ERROR_T := BYTE#01;
		state := 100;
	END_IF;

60:
	IF HTTP_GET.DONE THEN
		state := 80;
		CTRL.START_POS := HTTP_GET.BODY_START;
		CTRL.STOP_POS := HTTP_GET.BODY_STOP;
		CTRL.COMMAND := WORD#2#10000000_00011000; (* ONLY TEXT AND ATTRIBUTE *)
		CTRL.WATCHDOG := T#1ms;

	ELSIF (HTTP_GET.ERROR > DWORD#00) THEN
		(* Fehlerbehandlung *)
		ERROR_C := HTTP_GET.ERROR;
		ERROR_T := BYTE#02;
		state := 100;
	END_IF;

80:
	(* XML Daten seriell lesen *)
	XML_READER(CTRL:=CTRL,BUF:=R_BUF.BUFFER);
	IF CTRL.TYP < 98 THEN (* nur auswerten wenn kein Watchdog durchlauf *)
		(* automatische konvertierung in real und int ausführen *)
		value_int := 0;
		value_real := 0.0;
		IF LEN(CTRL.VALUE) <= 20 THEN
			v_real :=OSCAT_BASIC.FLOAT_TO_REAL(FLT:=CTRL.VALUE);
			IF OSCAT_BASIC.CHK_REAL(v_real) = 0 THEN (* !!! prüft auf gültigen REAL Wert, ansonsten stürzt Twincat ab !!!!  *)
				value_real := v_real;
				value_int := REAL_TO_INT(value_real);
			END_IF;
		END_IF;

		CASE UINT_TO_INT(CTRL.COUNT) OF

